# B&R Automation Studio project KeePakST401VersionX (part 3)

#### Types.typ - Exported data types
```iecst
TYPE
	DUT_NDSN_ADI : 	STRUCT
		ui_Size : UINT;
		ui_ADI : UINT;
	END_STRUCT;
	DUT_NDSN_Inventory : 	STRUCT
		b_r_TempCtrl_Board1 : BOOL;
		b_r_TempCtrl_Board2 : BOOL;
		b_r_TempCtrl_Board3 : BOOL;
		b_r_TempCtrl_Board4 : BOOL;
		b_r_OEM_Unit : BOOL;
		b_r_OLED_Unit : BOOL;
		b_r_WIFI_Board : BOOL;
		b_r_Refill_Board : BOOL;
		b_r_Anybus_Board : BOOL;
		b_r_Press_Sensor : BOOL;
		b_r_Press_CtrlValve : BOOL;
		i_r_NumOfTempZones_Internal : INT;
		i_r_NumOfTempZones_External : INT;
		i_r_NumOfMotors : INT;
		i_r_NumOfPumps : INT;
		i_r_NumOfATS : INT;
		i_r_NumOfWebClients : INT;
	END_STRUCT;
	DUT_NDSN_Flex : 	STRUCT
		b_r_SystemReady : BOOL;
		b_r_Fault : BOOL;
		b_r_Alert : BOOL;
		b_r_Stop : BOOL;
		b_r_LostCommunication : BOOL;
		b_w_ClearAlertFault : BOOL;
		b_r_TemperatureReady : BOOL;
		b_r_HeatersOn : BOOL;
		b_r_StandbyOn : BOOL;
		b_r_TemperatureAlert : BOOL;
		b_r_TemperatureFault : BOOL;
		b_r_PumpRunning : BOOL;
		b_r_PumpEnabled : BOOL;
		b_r_Purging : BOOL;
		b_r_TankLevelEmpty : BOOL;
		b_r_TankLevelLow : BOOL;
		b_r_FillSysAlert : BOOL;
		b_r_FillSysFault : BOOL;
		b_r_Filling : BOOL;
		b_r_LidOpen : BOOL;
		b_r_EmptyCalibrated : BOOL;
		b_w_HeatersOnOff : BOOL;
		b_w_StandbyOnOff : BOOL;
		b_w_PumpOnOff : BOOL;
		b_w_Purge : BOOL;
		b_w_ManualFill : BOOL;
		b_w_CalibrateEmpty : BOOL;
		b_w_CalibrateFull : BOOL;
		i_rw_Temp_arr_ZoneSP : ARRAY[0..17]OF INT;
		i_rw_Temp_arr_ZoneActivate : ARRAY[0..17]OF INT;
		i_rw_Temp_GlobalStandbyDelta : INT;
		i_rw_Temp_ManualStandyDuration : INT;
		i_rw_Temp_AutoEnterStandbyTm : INT;
		i_rw_Temp_AutoHeaterOffTime : INT;
		i_rw_Temp_AutoStandbySource : INT;
		i_rw_Temp_UnderTempDelta : INT;
		i_rw_Temp_OverTempDelta : INT;
		i_rw_Temp_Unit : INT;
		i_rw_Temp_GlobalSP : INT;
		i_rw_Temp_GlbalHoseSP : INT;
		i_rw_Temp_GlobalGunSP : INT;
		i_rw_Press_Unit : INT;
		r_rw_Press_SP : REAL;
		r_rw_Press_MaxPressLimit : REAL;
		r_rw_Press_MinPressLimit : REAL;
		r_rw_Press_UnderPressDelta : REAL;
		r_rw_Press_OverPressDelta : REAL;
		i_rw_Press_EnableHighLowAlert : INT;
		i_rw_Press_EnableHydrScale : INT;
		i_rw_Fill_EnableFill : INT;
		i_rw_Fill_TargetFillLevel : INT;
		i_rw_Fill_MaxFillTime : INT;
		i_rw_Fill_AlertStopDelayTime : INT;
		i_rw_Fill_LowLevelThreshold : INT;
		i_rw_Fill_LidOpenAlertTime : INT;
		i_rw_Fill_EmptyStopOnOff : INT;
		i_rw_Pump_AutoPump : INT;
		i_rw_Gen_ReadyDelayTime : INT;
		i_rw_Gen_MassUnit : INT;
		i_r_Temp_arr_ZoneActual : ARRAY[0..17]OF INT;
		i_r_Temp_arr_ZoneStatus : ARRAY[0..17]OF INT;
		r_r_Press_ActualPressure : REAL;
		i_r_Press_SensorAlarm : INT;
		i_r_Fill_TankLevel : INT;
		i_r_Gen_CurrentFaultCode : INT;
		i_r_Gen_SoftwareVersion : INT;
		di_r_Gen_OperationHrs : DINT;
		i_r_Gen_arr_SysInventory : ARRAY[0..3]OF INT;
		st_r_Devices : DUT_NDSN_Inventory;
	END_STRUCT;
END_TYPE
```

#### Lib_PBFlx.fun - Exported functions and function blocks
```iecst
{REDUND_OK} FUNCTION_BLOCK FB_NDSN_MB_PBFlex_CtrlSts (*ProblueFlex Function Block for ModbusTCP _Control& Status*) (*$GROUP=User,$CAT=User,$GROUPICON=User.png,$CATICON=User.png*)
	VAR_INPUT
		IN_b_Enable : {REDUND_UNREPLICABLE} BOOL;
		IN_mb_station : STRING[30];
	END_VAR
	VAR_IN_OUT
		Melter : DUT_NDSN_Flex;
	END_VAR
	VAR
		IO_Input : ARRAY[0..63] OF UINT;
		IO_Output : ARRAY[0..63] OF UINT;
		tm_HeaterOff : TON;
		b_HeaterOff : BOOL;
		b_Temp1 : BOOL;
		b_Temp2 : BOOL;
		b_Temp3 : BOOL;
		b_Temp4 : BOOL;
		b_HeaterOn : BOOL;
		tm_HeaterOnStuck : TON;
		b_HeaterOnStuck : BOOL;
		tm_HeaterOffStuck : TON;
		b_HeaterOffStuck : BOOL;
		tm_PumpOff : TON;
		b_PumpOff : BOOL;
		tm_PumpOnStuck : TON;
		b_PumpOnStuck : BOOL;
		tm_PumpOffStuck : TON;
		b_PumpOffStuck : BOOL;
		tm_StandbyOff : TON;
		b_StandbyOff : BOOL;
		tm_StandbyOnStuck : TON;
		b_StandbyOnStuck : BOOL;
		tm_StandbyOffStuck : TON;
		b_StandbyOffStuck : BOOL;
		b_Temp5 : BOOL;
		b_Temp6 : BOOL;
		b_StandbyOn : BOOL;
		b_PumpOn : BOOL;
		tm_Command : TON;
		b_CommandTimerRising : BOOL;
		b_Init : BOOL;
		tm_Acyc : TON;
		b_read : BOOL;
		ui_AcycRdStatus : UINT;
		i : INT;
		FB_AcycWrite : mbWriteMultipleRegisters;
		FB_AcycRead : mbReadHoldingRegisters;
		ui_AcycWtStatus : UINT;
		i_StartAddressOutput : INT;
		i_StartAddressInput : INT;
		i_datasize : INT;
		i_nrRegisters : UINT;
	END_VAR
END_FUNCTION_BLOCK

{REDUND_OK} FUNCTION_BLOCK FB_NDSN_MB_PBFlex_Process (*ProblueFlex Function Block for ModbusTCP _Process*) (*$GROUP=User,$CAT=User,$GROUPICON=User.png,$CATICON=User.png*)
	VAR_INPUT
		IN_b_Enable : {REDUND_UNREPLICABLE} BOOL;
		IN_mb_station : STRING[30];
	END_VAR
	VAR_IN_OUT
		Melter : DUT_NDSN_Flex;
	END_VAR
	VAR
		IO_Input : ARRAY[0..63] OF UINT;
		IO_Output : ARRAY[0..63] OF UINT;
		b_Init : BOOL;
		tm_Acyc : TON;
		b_read : BOOL;
		st_ADI_List : ARRAY[0..49] OF DUT_NDSN_ADI;
		b_AcycRD_Enable : BOOL;
		b_AcycRD_Done : BOOL;
		b_AcycRD_Tick : BOOL;
		ui_AcycRdStatus_Para : UINT;
		ui_AcycRdStatus : UINT;
		b_AcycRdDnRising : BOOL;
		i : INT;
		arr_ResponseValue : ARRAY[0..17] OF UINT;
		i_ValueIndex : INT;
		i_rwDataSize : INT := 70;
		arr_HMI : ARRAY[0..119] OF UINT;
		arr_HMI_Buffer : ARRAY[0..69] OF UINT;
		arr_HMI_Compare : ARRAY[0..69] OF UINT;
		b_WriteEvent : BOOL;
		arr_WriteIndex : ARRAY[0..30] OF INT;
		i_rwADI_Count : INT := 30;
		i_ADI_Range : INT;
		FB_AcycWrite : mbWriteMultipleRegisters;
		FB_AcycRead_Para : mbReadHoldingRegisters;
		i_ADI_Size : INT := 40;
		i_Index : INT;
		i_Index_Write : INT;
		arr_WriteStartingAddress : ARRAY[0..31] OF INT;
		i_ADI : INT;
		di_Press : UDINT;
		di_Press_psi : UDINT;
		r_Press : REAL;
		r_PressConvert : REAL;
		arr_i_DW_Temp : ARRAY[0..1] OF UINT;
		arr_di_Press_psi : ARRAY[0..1] OF UINT;
		tm_WriteEvent : TON;
		i_CompareIndex : INT;
		b_AcycWT_Done : BOOL;
		b_WriteEventONS : BOOL;
		i_writesize : INT;
		i_arr_WriteBuffer : ARRAY[0..17] OF INT;
		i_Size : INT;
		i_SizeofStruct : INT := 236;
		b_Temp2 : BOOL;
		b_AcycWT_DN_Rising : BOOL;
		b_AcycWT_Start : BOOL;
		b_AcycWT_Rising : BOOL;
		ui_AcycWtStatus : UINT;
		i_wttest : UINT;
		b_AcycWTDnRising : BOOL;
		b_test : BOOL;
		i_StartAddressOutput : INT;
		i_StartAddressInput : INT;
		i_datasize : INT;
		ui_Compare : UINT;
		ui_Ctrl : UINT;
		b_temp1 : BOOL;
		b_Compare : BOOL;
		tm_Compare : TON;
		i_test : INT;
		i_nrRegisters : UINT;
	END_VAR
END_FUNCTION_BLOCK
```

### Program Logical/Simulation/Simulation (IEC)

#### Variables.var
```iecst
VAR
	TON_Test : TON;
END_VAR
```

#### Main.st
```iecst
PROGRAM _INIT

	gIO.DIs.SafetyOK := TRUE;
	gIO.SafetyStatus.SafetyProgramRunning := TRUE;

		TON_Test.PT := T#300ms;

END_PROGRAM

PROGRAM _CYCLIC

	//DetermineDistanceToStopPos(gIO.Encoders.SickSSIPosDegrees,

	TON_Test.IN := NOT TON_Test.Q;
//	TON_Test.PT := T#100ms;
	IF EDGEPOS(TON_Test.Q) THEN
		gIO.Encoders.SickSSIPosDegrees := gIO.Encoders.SickSSIPosDegrees + 1;
	END_IF
	IF (gIO.Encoders.SickSSIPosDegrees > 360) THEN
		gIO.Encoders.SickSSIPosDegrees := 0;
	END_IF
	TON_Test();

END_PROGRAM
```

### Program Logical/ModeControl/ModeControl (IEC) - Copy right:KeePak, B&R  Authors: Nathan Stephens, Jeremy Lee, Cody Jung   Rev:1.0   Date:9-28-17

#### Cyclic.ld - Cyclic code
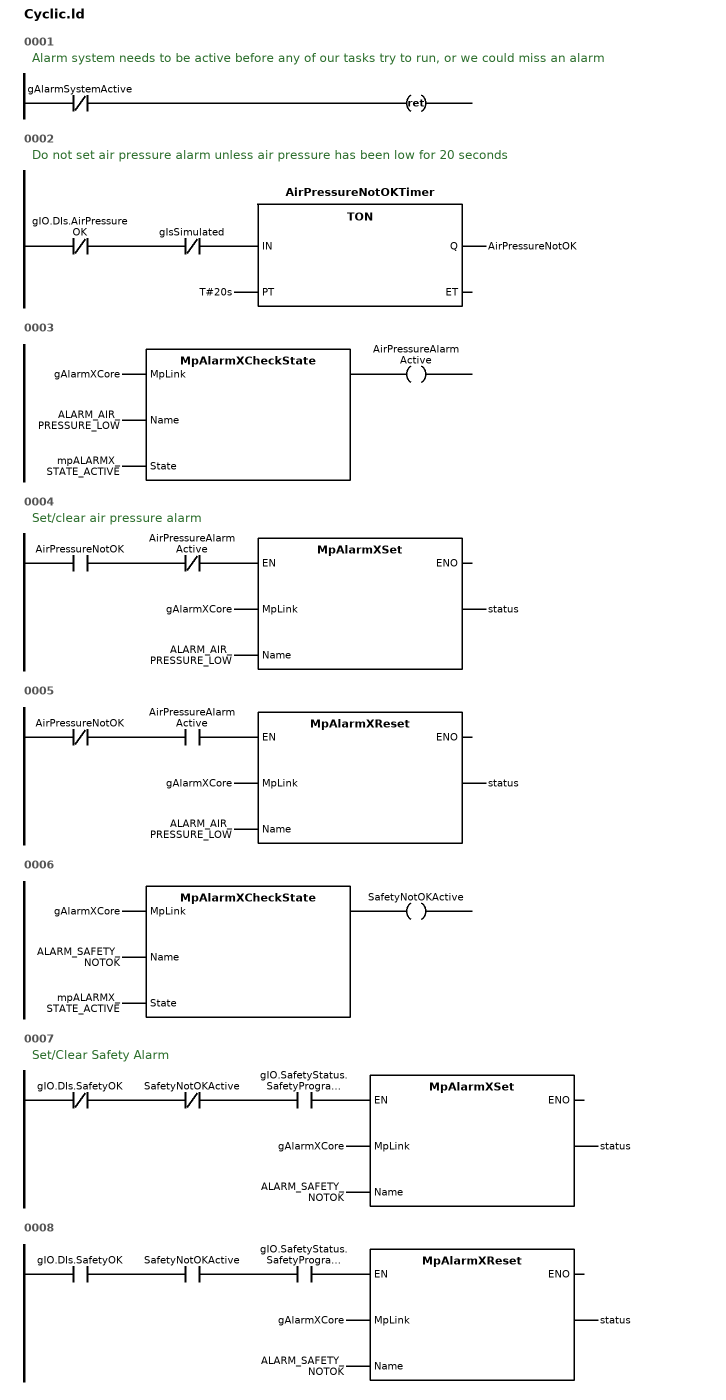
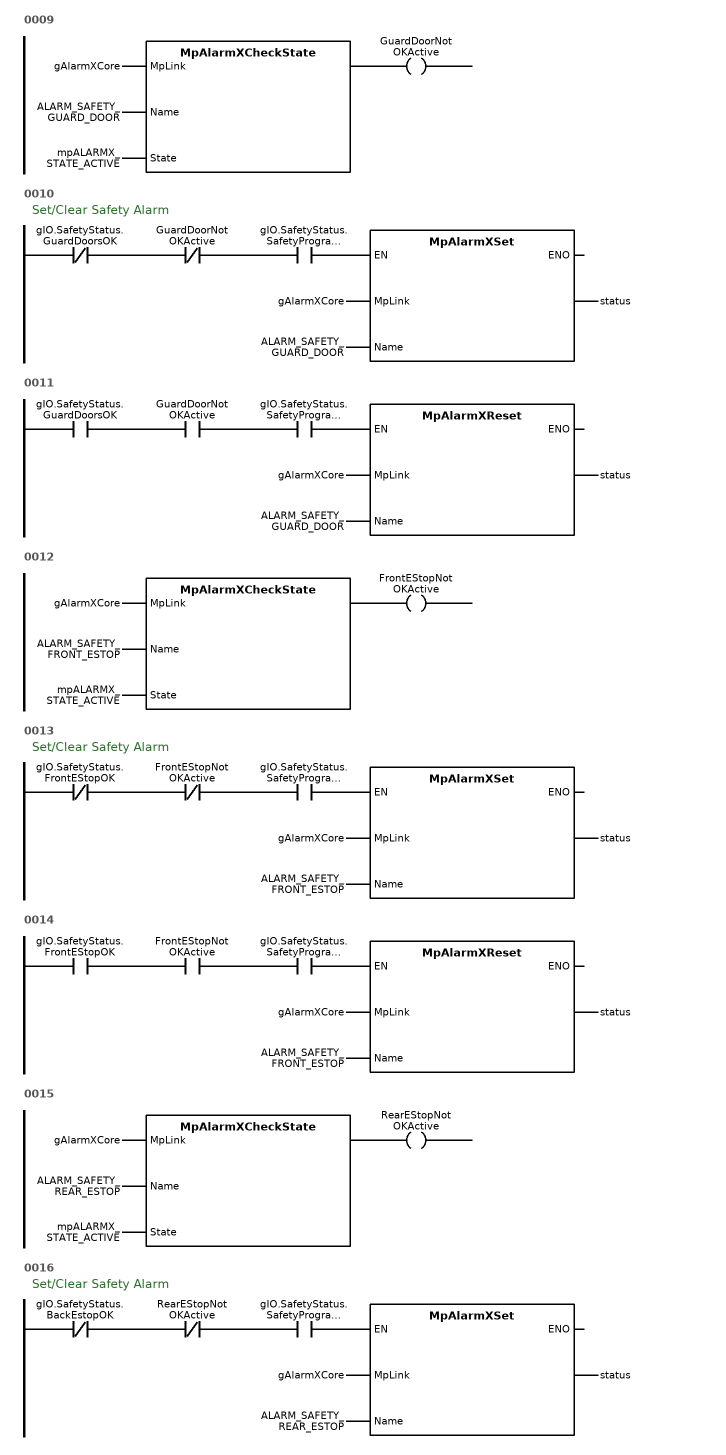
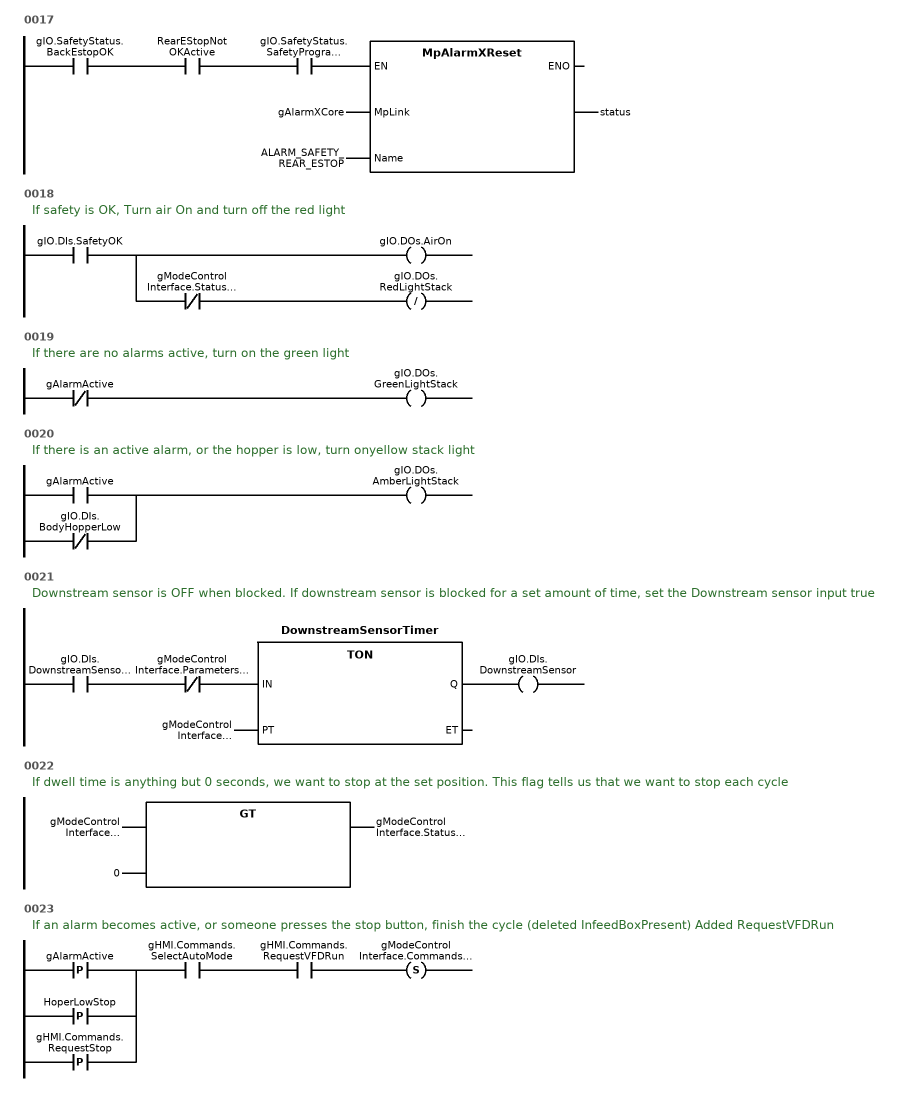
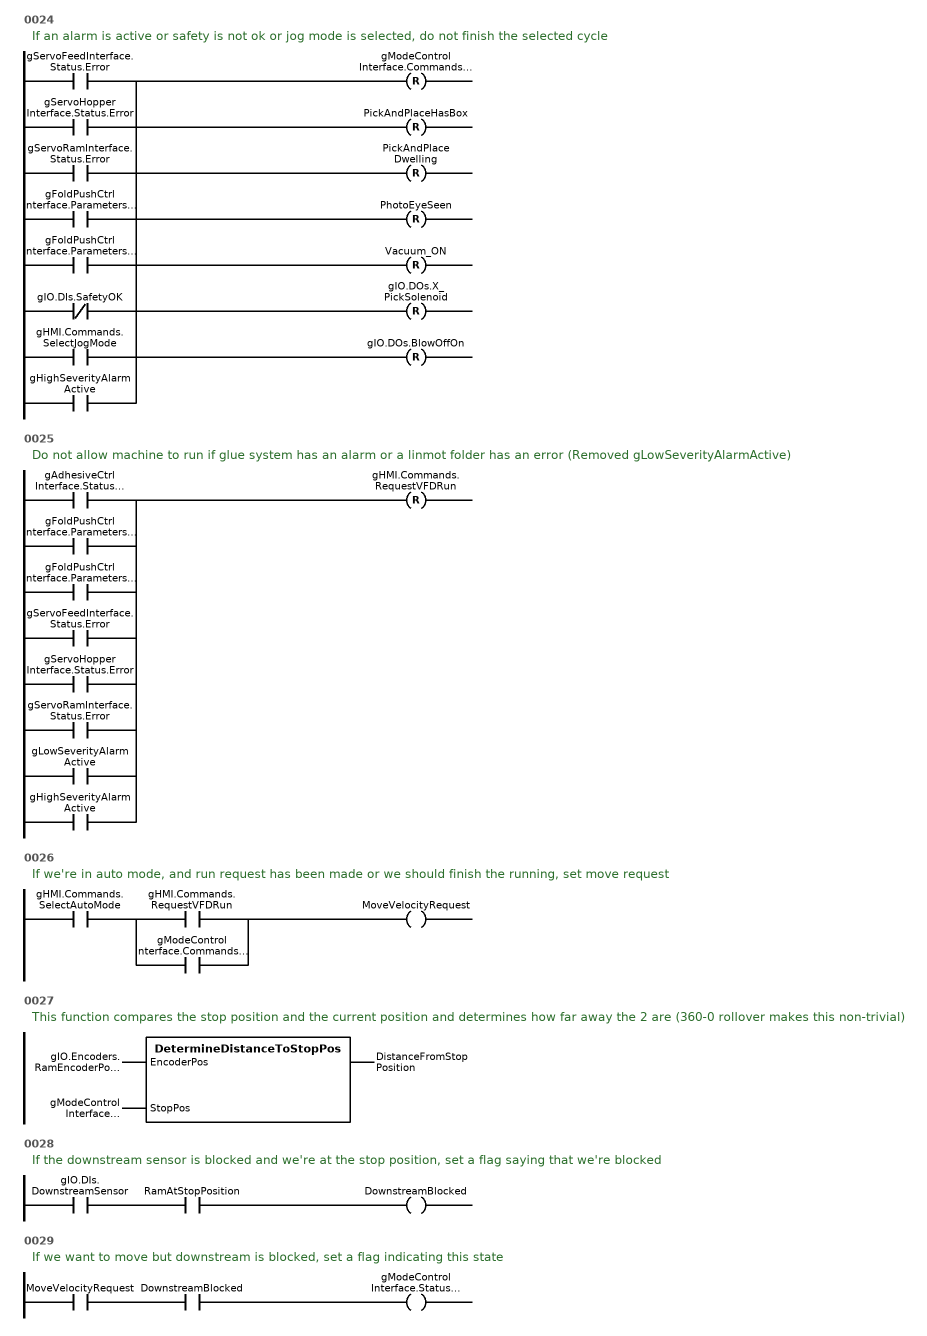
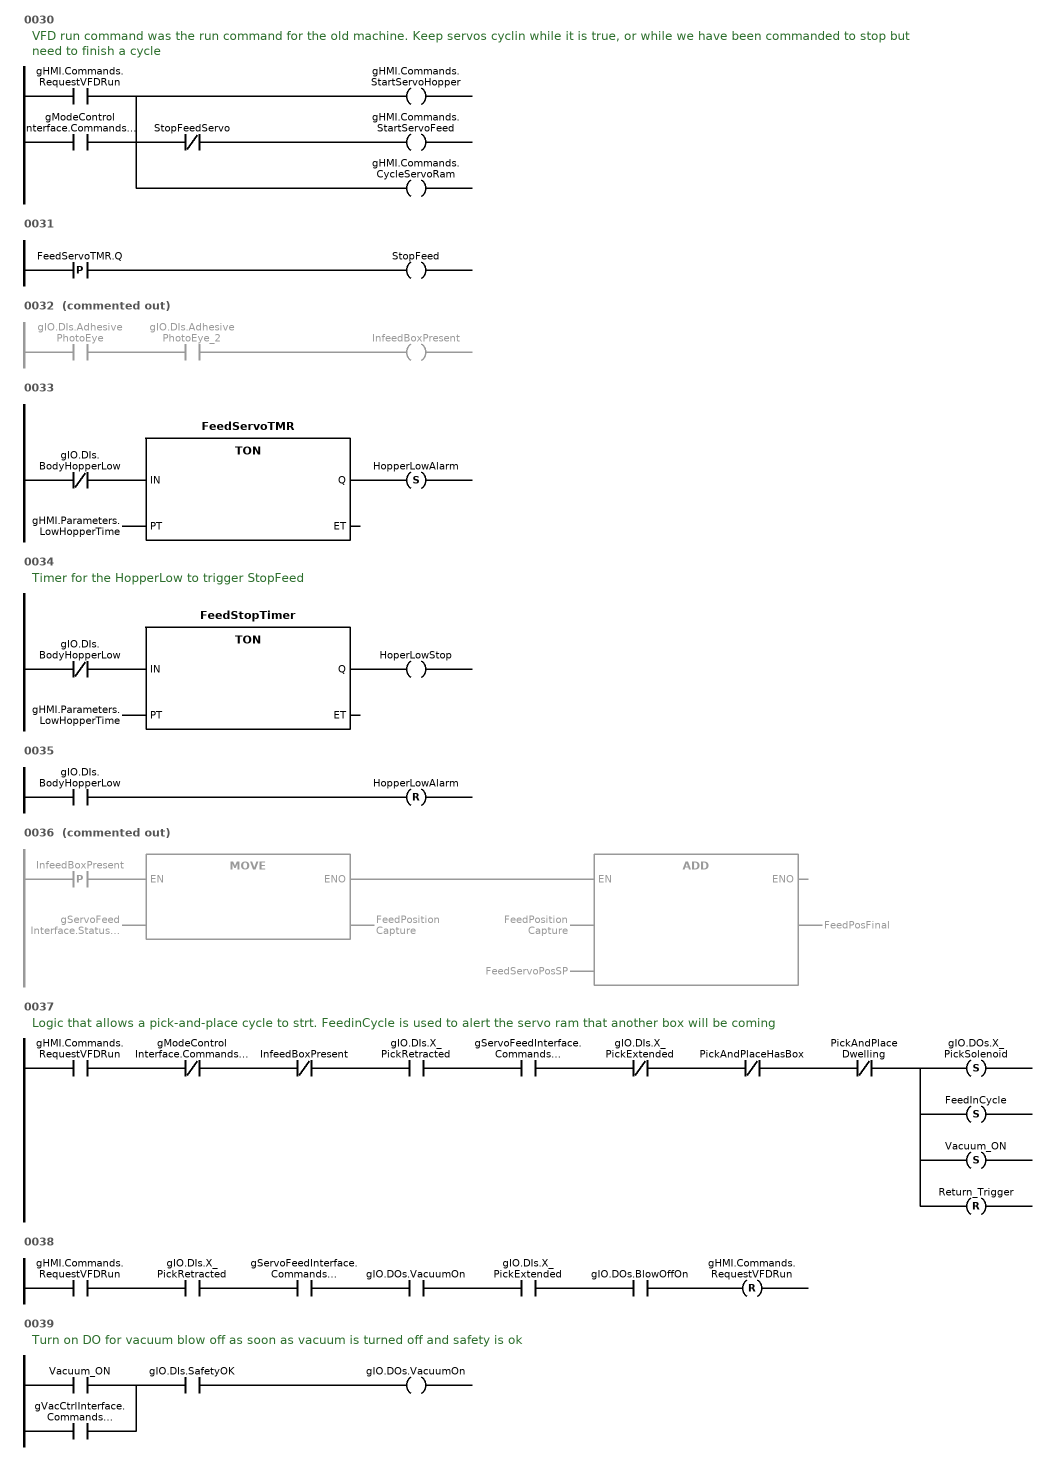
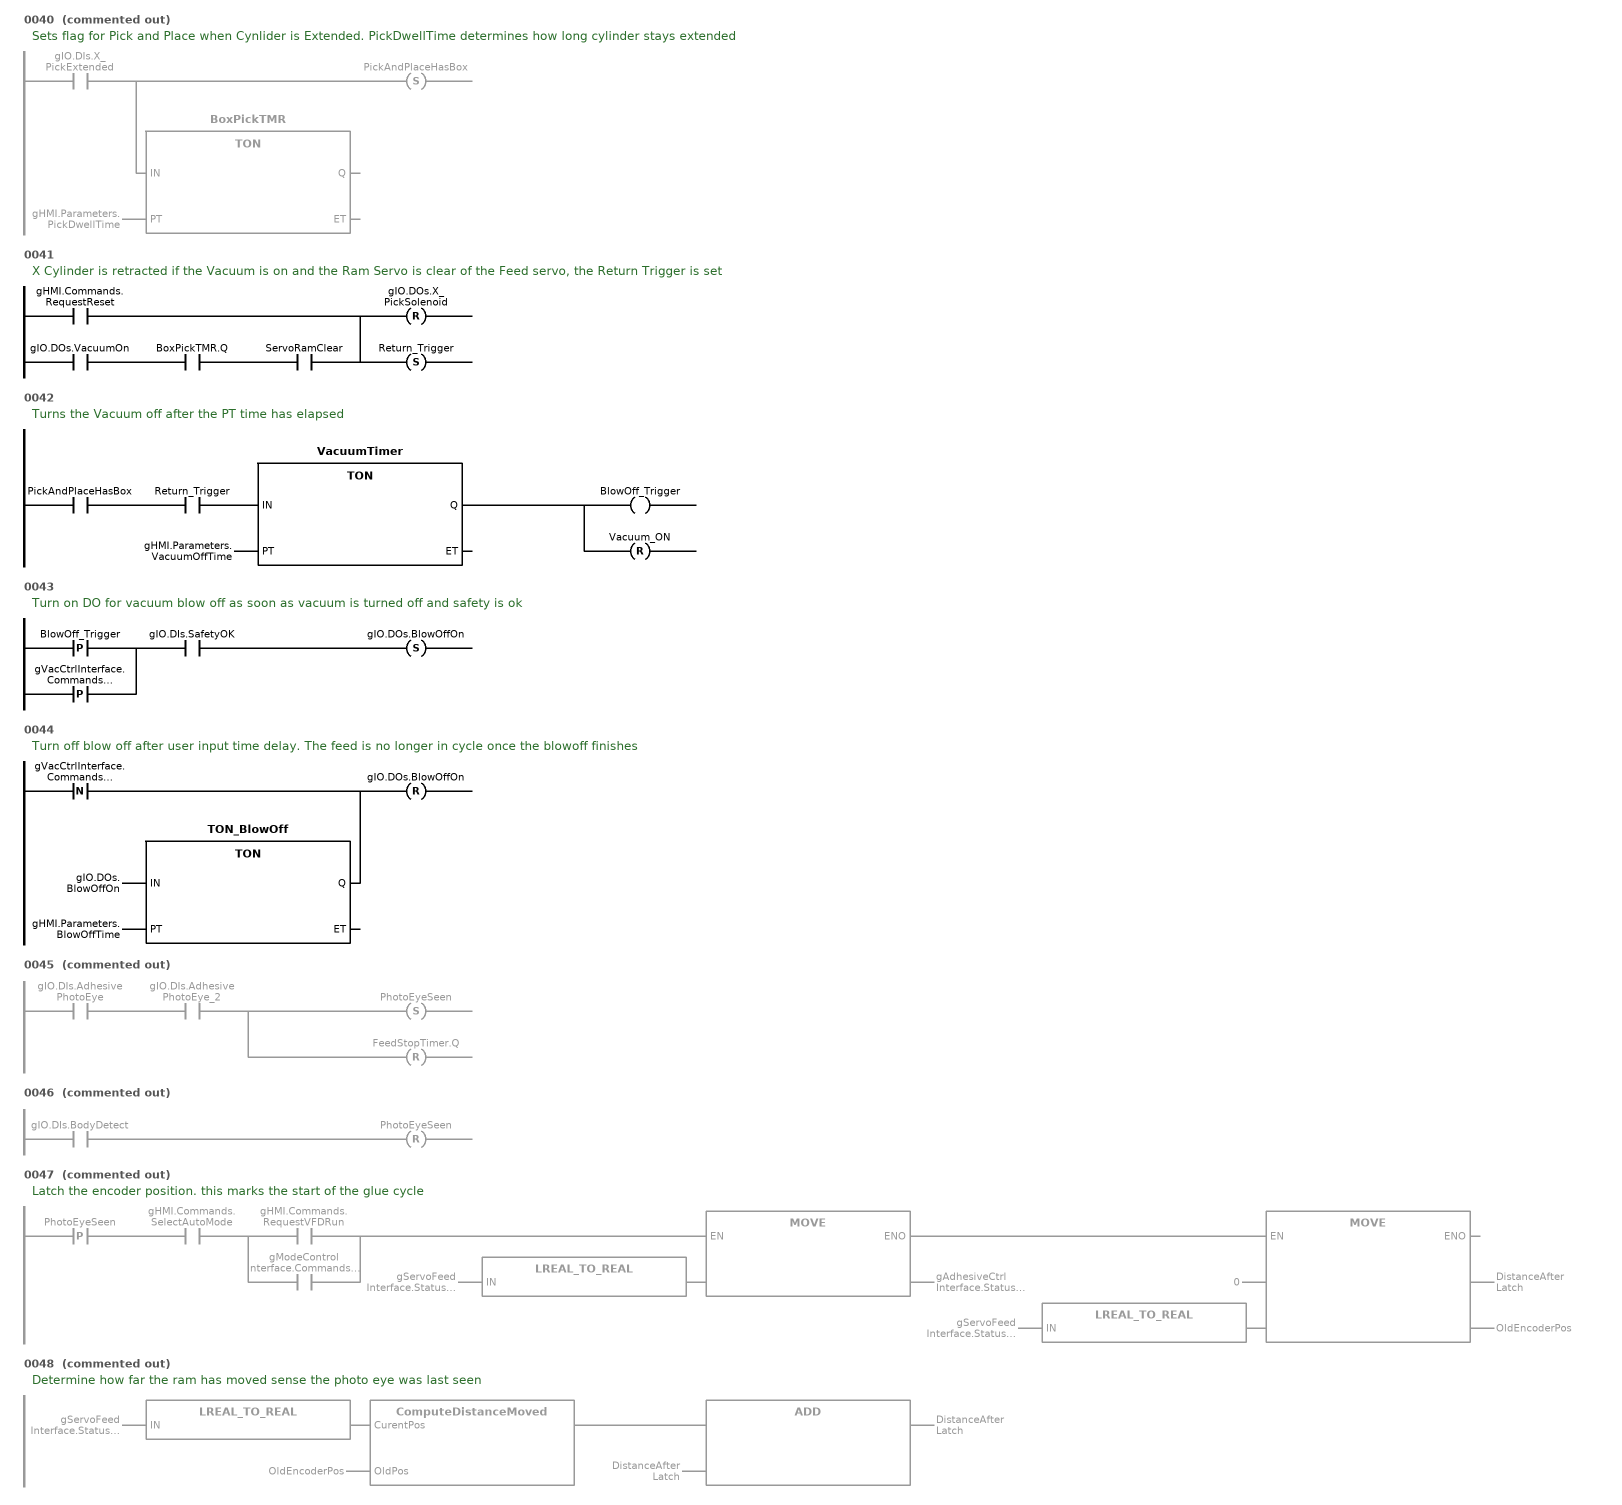
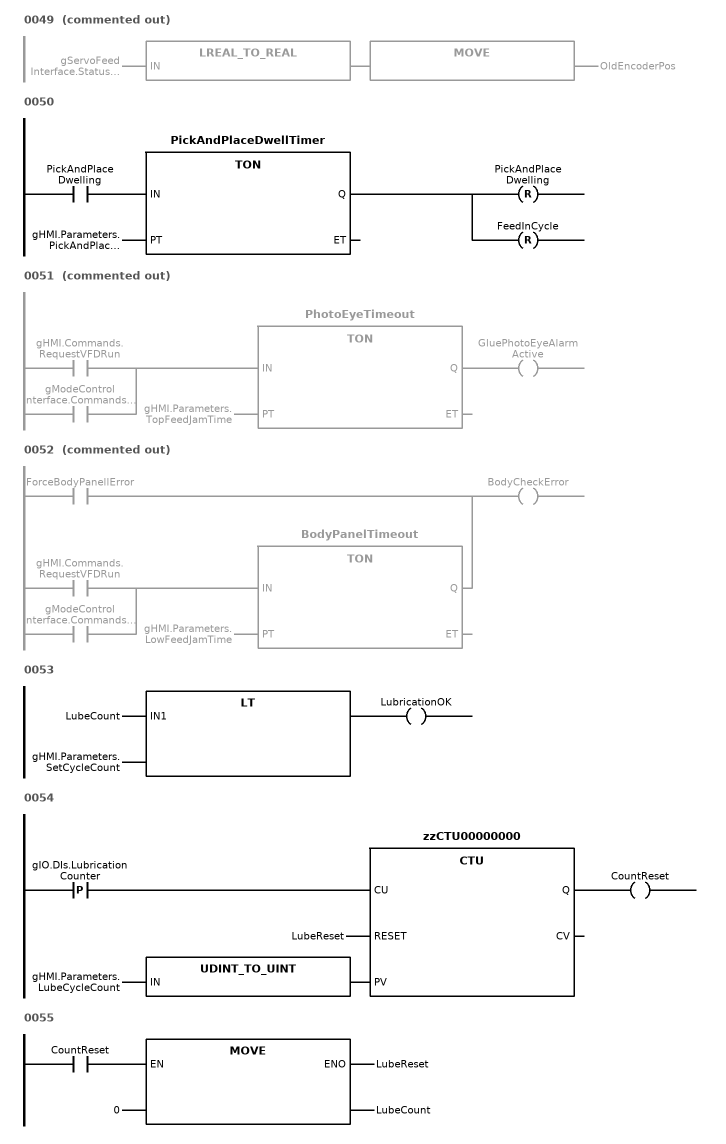
Ladder, written as Structured Text:
```iecst
PROGRAM _CYCLIC
VAR
    _p1 : BOOL;
    _e2 : R_TRIG;
    _e3 : R_TRIG;
    _e4 : R_TRIG;
    _p5 : BOOL;
    _p6 : BOOL;
    _p7 : BOOL;
    _p8 : BOOL;
    _e9 : R_TRIG;
    _e10 : R_TRIG;
    _p11 : BOOL;
    _p12 : BOOL;
    _e13 : R_TRIG;
    _e14 : R_TRIG;
    _e15 : F_TRIG;
    _p16 : BOOL;
    _e17 : R_TRIG;
    _e18 : R_TRIG;
END_VAR
(* Network 1: Alarm system needs to be active before any of our tasks try to run, or we could miss an alarm *)
IF NOT gAlarmSystemActive THEN RETURN; END_IF;

(* Network 2: Do not set air pressure alarm unless air pressure has been low for 20 seconds *)
AirPressureNotOKTimer(IN := NOT gIO.DIs.AirPressureOK AND NOT gIsSimulated, PT := T#20s);
AirPressureNotOK := AirPressureNotOKTimer.Q;

(* Network 3 *)
AirPressureAlarmActive := MpAlarmXCheckState(MpLink := gAlarmXCore, Name := ALARM_AIR_PRESSURE_LOW, State := mpALARMX_STATE_ACTIVE);

(* Network 4: Set/clear air pressure alarm *)
IF AirPressureNotOK AND NOT AirPressureAlarmActive THEN
    status := MpAlarmXSet(MpLink := gAlarmXCore, Name := ALARM_AIR_PRESSURE_LOW);
END_IF;

(* Network 5 *)
IF NOT AirPressureNotOK AND AirPressureAlarmActive THEN
    status := MpAlarmXReset(MpLink := gAlarmXCore, Name := ALARM_AIR_PRESSURE_LOW);
END_IF;

(* Network 6 *)
SafetyNotOKActive := MpAlarmXCheckState(MpLink := gAlarmXCore, Name := ALARM_SAFETY_NOTOK, State := mpALARMX_STATE_ACTIVE);

(* Network 7: Set/Clear Safety Alarm *)
IF NOT gIO.DIs.SafetyOK AND NOT SafetyNotOKActive AND gIO.SafetyStatus.SafetyProgramRunning THEN
    status := MpAlarmXSet(MpLink := gAlarmXCore, Name := ALARM_SAFETY_NOTOK);
END_IF;

(* Network 8 *)
IF gIO.DIs.SafetyOK AND SafetyNotOKActive AND gIO.SafetyStatus.SafetyProgramRunning THEN
    status := MpAlarmXReset(MpLink := gAlarmXCore, Name := ALARM_SAFETY_NOTOK);
END_IF;

(* Network 9 *)
GuardDoorNotOKActive := MpAlarmXCheckState(MpLink := gAlarmXCore, Name := ALARM_SAFETY_GUARD_DOOR, State := mpALARMX_STATE_ACTIVE);

(* Network 10: Set/Clear Safety Alarm *)
IF NOT gIO.SafetyStatus.GuardDoorsOK AND NOT GuardDoorNotOKActive AND gIO.SafetyStatus.SafetyProgramRunning THEN
    status := MpAlarmXSet(MpLink := gAlarmXCore, Name := ALARM_SAFETY_GUARD_DOOR);
END_IF;

(* Network 11 *)
IF gIO.SafetyStatus.GuardDoorsOK AND GuardDoorNotOKActive AND gIO.SafetyStatus.SafetyProgramRunning THEN
    status := MpAlarmXReset(MpLink := gAlarmXCore, Name := ALARM_SAFETY_GUARD_DOOR);
END_IF;

(* Network 12 *)
FrontEStopNotOKActive := MpAlarmXCheckState(MpLink := gAlarmXCore, Name := ALARM_SAFETY_FRONT_ESTOP, State := mpALARMX_STATE_ACTIVE);

(* Network 13: Set/Clear Safety Alarm *)
IF NOT gIO.SafetyStatus.FrontEStopOK AND NOT FrontEStopNotOKActive AND gIO.SafetyStatus.SafetyProgramRunning THEN
    status := MpAlarmXSet(MpLink := gAlarmXCore, Name := ALARM_SAFETY_FRONT_ESTOP);
END_IF;

(* Network 14 *)
IF gIO.SafetyStatus.FrontEStopOK AND FrontEStopNotOKActive AND gIO.SafetyStatus.SafetyProgramRunning THEN
    status := MpAlarmXReset(MpLink := gAlarmXCore, Name := ALARM_SAFETY_FRONT_ESTOP);
END_IF;

(* Network 15 *)
RearEStopNotOKActive := MpAlarmXCheckState(MpLink := gAlarmXCore, Name := ALARM_SAFETY_REAR_ESTOP, State := mpALARMX_STATE_ACTIVE);

(* Network 16: Set/Clear Safety Alarm *)
IF NOT gIO.SafetyStatus.BackEstopOK AND NOT RearEStopNotOKActive AND gIO.SafetyStatus.SafetyProgramRunning THEN
    status := MpAlarmXSet(MpLink := gAlarmXCore, Name := ALARM_SAFETY_REAR_ESTOP);
END_IF;

(* Network 17 *)
IF gIO.SafetyStatus.BackEstopOK AND RearEStopNotOKActive AND gIO.SafetyStatus.SafetyProgramRunning THEN
    status := MpAlarmXReset(MpLink := gAlarmXCore, Name := ALARM_SAFETY_REAR_ESTOP);
END_IF;

(* Network 18: If safety is OK, Turn air On and turn off the red light *)
_p1 := gIO.DIs.SafetyOK;
gIO.DOs.AirOn := gIO.DIs.SafetyOK;
gIO.DOs.RedLightStack := NOT (_p1 AND NOT gModeControlInterface.Status.BlissPanelAlarmActive);

(* Network 19: If there are no alarms active, turn on the green light *)
gIO.DOs.GreenLightStack := NOT gAlarmActive;

(* Network 20: If there is an active alarm, or the hopper is low, turn onyellow stack light *)
gIO.DOs.AmberLightStack := gAlarmActive OR NOT gIO.DIs.BodyHopperLow;

(* Network 21: Downstream sensor is OFF when blocked. If downstream sensor is blocked for a set amount of time, set the Downstream sensor input true *)
DownstreamSensorTimer(IN := gIO.DIs.DownstreamSensorRaw AND NOT gModeControlInterface.Parameters.DownstreamIgnored, PT := gModeControlInterface.Parameters.DownstreamTimeout);
gIO.DIs.DownstreamSensor := DownstreamSensorTimer.Q;

(* Network 22: If dwell time is anything but 0 seconds, we want to stop at the set position. This flag tells us that we want to stop each cycle *)
gModeControlInterface.Status.DwellModeEnabled := gModeControlInterface.Parameters.DwellTime > 0;

(* Network 23: If an alarm becomes active, or someone presses the stop button, finish the cycle (deleted InfeedBoxPresent) Added RequestVFDRun *)
_e2(CLK := gAlarmActive);
_e3(CLK := HoperLowStop);
_e4(CLK := gHMI.Commands.RequestStop);
IF (_e2.Q OR _e3.Q OR _e4.Q) AND gHMI.Commands.SelectAutoMode AND gHMI.Commands.RequestVFDRun THEN
    gModeControlInterface.Commands.FinishCycle := TRUE;
END_IF;

(* Network 24: If an alarm is active or safety is not ok or jog mode is selected, do not finish the selected cycle *)
_p5 := gFoldPushCtrlInterface.Parameters.LinMotBotFolder.Status.Error;
_p6 := gFoldPushCtrlInterface.Parameters.LinMotTopFolder.Status.Error;
IF gServoFeedInterface.Status.Error OR gServoHopperInterface.Status.Error OR gServoRamInterface.Status.Error OR _p5 OR _p6 OR NOT gIO.DIs.SafetyOK OR gHMI.Commands.SelectJogMode OR gHighSeverityAlarmActive THEN
    gModeControlInterface.Commands.FinishCycle := FALSE;
    PickAndPlaceHasBox := FALSE;
    PickAndPlaceDwelling := FALSE;
    PhotoEyeSeen := FALSE;
    Vacuum_ON := FALSE;
END_IF;
_p7 := NOT gIO.DIs.SafetyOK;
IF gServoFeedInterface.Status.Error OR gServoHopperInterface.Status.Error OR gServoRamInterface.Status.Error OR _p5 OR _p6 OR NOT gIO.DIs.SafetyOK OR gHMI.Commands.SelectJogMode OR gHighSeverityAlarmActive THEN
    gIO.DOs.X_PickSolenoid := FALSE;
END_IF;
IF gServoFeedInterface.Status.Error OR gServoHopperInterface.Status.Error OR gServoRamInterface.Status.Error OR _p5 OR _p6 OR _p7 OR gHMI.Commands.SelectJogMode OR gHighSeverityAlarmActive THEN
    gIO.DOs.BlowOffOn := FALSE;
END_IF;

(* Network 25: Do not allow machine to run if glue system has an alarm or a linmot folder has an error (Removed gLowSeverityAlarmActive) *)
IF gAdhesiveCtrlInterface.Status.AlarmActive OR gFoldPushCtrlInterface.Parameters.LinMotBotFolder.Status.Error OR gFoldPushCtrlInterface.Parameters.LinMotTopFolder.Status.Error OR gServoFeedInterface.Status.Error OR gServoHopperInterface.Status.Error OR gServoRamInterface.Status.Error OR gLowSeverityAlarmActive OR gHighSeverityAlarmActive THEN
    gHMI.Commands.RequestVFDRun := FALSE;
END_IF;

(* Network 26: If we're in auto mode, and run request has been made or we should finish the running, set move request *)
MoveVelocityRequest := gHMI.Commands.SelectAutoMode AND (gHMI.Commands.RequestVFDRun OR gModeControlInterface.Commands.FinishCycle);

(* Network 27: This function compares the stop position and the current position and determines how far away the 2 are (360-0 rollover makes this non-trivial) *)
DistanceFromStopPosition := DetermineDistanceToStopPos(EncoderPos := gIO.Encoders.RamEncoderPosDegrees, StopPos := gModeControlInterface.Parameters.StopPosition);

(* Network 28: If the downstream sensor is blocked and we're at the stop position, set a flag saying that we're blocked *)
DownstreamBlocked := gIO.DIs.DownstreamSensor AND RamAtStopPosition;

(* Network 29: If we want to move but downstream is blocked, set a flag indicating this state *)
gModeControlInterface.Status.WaitingOnDownstream := MoveVelocityRequest AND DownstreamBlocked;

(* Network 30: VFD run command was the run command for the old machine. Keep servos cyclin while it is true, or while we have been commanded to stop but need to finish a cycle *)
_p8 := gHMI.Commands.RequestVFDRun;
gHMI.Commands.StartServoHopper := gHMI.Commands.RequestVFDRun OR gModeControlInterface.Commands.FinishCycle;
gHMI.Commands.StartServoFeed := (_p8 OR gModeControlInterface.Commands.FinishCycle) AND NOT StopFeedServo;
gHMI.Commands.CycleServoRam := _p8 OR gModeControlInterface.Commands.FinishCycle;

(* Network 31 *)
_e9(CLK := FeedServoTMR.Q);
StopFeed := _e9.Q;

(* Network 32 *) (* commented out *)
// InfeedBoxPresent := gIO.DIs.AdhesivePhotoEye AND gIO.DIs.AdhesivePhotoEye_2;

(* Network 33 *)
FeedServoTMR(IN := NOT gIO.DIs.BodyHopperLow, PT := gHMI.Parameters.LowHopperTime);
IF FeedServoTMR.Q THEN HopperLowAlarm := TRUE; END_IF;

(* Network 34: Timer for the HopperLow to trigger StopFeed *)
FeedStopTimer(IN := NOT gIO.DIs.BodyHopperLow, PT := gHMI.Parameters.LowHopperTime);
HoperLowStop := FeedStopTimer.Q;

(* Network 35 *)
IF gIO.DIs.BodyHopperLow THEN HopperLowAlarm := FALSE; END_IF;

(* Network 36 *) (* commented out *)
// _e10(CLK := InfeedBoxPresent);
// IF _e10.Q THEN
//     FeedPositionCapture := gServoFeedInterface.Status.ActualPosition;
//     FeedPosFinal := FeedPositionCapture + FeedServoPosSP;
// END_IF;

(* Network 37: Logic that allows a pick-and-place cycle to strt. FeedinCycle is used to alert the servo ram that another box will be coming *)
_p11 := gHMI.Commands.RequestVFDRun AND NOT gModeControlInterface.Commands.FinishCycle AND NOT InfeedBoxPresent AND gIO.DIs.X_PickRetracted AND gServoFeedInterface.Commands.RequestMoveVelocity AND NOT gIO.DIs.X_PickExtended AND NOT PickAndPlaceHasBox AND NOT PickAndPlaceDwelling;
IF _p11 THEN
    gIO.DOs.X_PickSolenoid := TRUE;
    FeedInCycle := TRUE;
    Vacuum_ON := TRUE;
    Return_Trigger := FALSE;
END_IF;

(* Network 38 *)
IF gHMI.Commands.RequestVFDRun AND gIO.DIs.X_PickRetracted AND gServoFeedInterface.Commands.RequestMoveVelocity AND gIO.DOs.VacuumOn AND gIO.DIs.X_PickExtended AND gIO.DOs.BlowOffOn THEN
    gHMI.Commands.RequestVFDRun := FALSE;
END_IF;

(* Network 39: Turn on DO for vacuum blow off as soon as vacuum is turned off and safety is ok *)
gIO.DOs.VacuumOn := (Vacuum_ON OR gVacCtrlInterface.Commands.VenturiOnManual) AND gIO.DIs.SafetyOK;

(* Network 40: Sets flag for Pick and Place when Cynlider is Extended. PickDwellTime determines how long cylinder stays extended *) (* commented out *)
// IF gIO.DIs.X_PickExtended THEN PickAndPlaceHasBox := TRUE; END_IF;
// BoxPickTMR(IN := gIO.DIs.X_PickExtended, PT := gHMI.Parameters.PickDwellTime);

(* Network 41: X Cylinder is retracted if the Vacuum is on and the Ram Servo is clear of the Feed servo, the Return Trigger is set *)
_p12 := gIO.DOs.VacuumOn AND BoxPickTMR.Q AND ServoRamClear;
IF gHMI.Commands.RequestReset OR _p12 THEN
    gIO.DOs.X_PickSolenoid := FALSE;
    Return_Trigger := TRUE;
END_IF;

(* Network 42: Turns the Vacuum off after the PT time has elapsed *)
VacuumTimer(IN := PickAndPlaceHasBox AND Return_Trigger, PT := gHMI.Parameters.VacuumOffTime);
BlowOff_Trigger := VacuumTimer.Q;
IF VacuumTimer.Q THEN Vacuum_ON := FALSE; END_IF;

(* Network 43: Turn on DO for vacuum blow off as soon as vacuum is turned off and safety is ok *)
_e13(CLK := BlowOff_Trigger);
_e14(CLK := gVacCtrlInterface.Commands.BlowOffOnManual);
IF (_e13.Q OR _e14.Q) AND gIO.DIs.SafetyOK THEN gIO.DOs.BlowOffOn := TRUE; END_IF;

(* Network 44: Turn off blow off after user input time delay. The feed is no longer in cycle once the blowoff finishes *)
_e15(CLK := gVacCtrlInterface.Commands.BlowOffOnManual);
IF _e15.Q OR TON_BlowOff.Q THEN gIO.DOs.BlowOffOn := FALSE; END_IF;
TON_BlowOff(IN := gIO.DOs.BlowOffOn, PT := gHMI.Parameters.BlowOffTime);

(* Network 45 *) (* commented out *)
// _p16 := gIO.DIs.AdhesivePhotoEye AND gIO.DIs.AdhesivePhotoEye_2;
// IF _p16 THEN
//     PhotoEyeSeen := TRUE;
//     FeedStopTimer.Q := FALSE;
// END_IF;

(* Network 46 *) (* commented out *)
// IF gIO.DIs.BodyDetect THEN PhotoEyeSeen := FALSE; END_IF;

(* Network 47: Latch the encoder position. this marks the start of the glue cycle *) (* commented out *)
// _e17(CLK := PhotoEyeSeen);
// IF _e17.Q AND gHMI.Commands.SelectAutoMode AND (gHMI.Commands.RequestVFDRun OR gModeControlInterface.Commands.FinishCycle) THEN
//     gAdhesiveCtrlInterface.Status.LatchedEncoderPos := LREAL_TO_REAL(gServoFeedInterface.Status.ActualPosition);
//     DistanceAfterLatch := 0;
//     OldEncoderPos := LREAL_TO_REAL(gServoFeedInterface.Status.ActualPosition);
// END_IF;

(* Network 48: Determine how far the ram has moved sense the photo eye was last seen *) (* commented out *)
// DistanceAfterLatch := ComputeDistanceMoved(CurentPos := LREAL_TO_REAL(gServoFeedInterface.Status.ActualPosition), OldPos := OldEncoderPos) + DistanceAfterLatch;

(* Network 49 *) (* commented out *)
// OldEncoderPos := LREAL_TO_REAL(gServoFeedInterface.Status.ActualPosition);

(* Network 50 *)
PickAndPlaceDwellTimer(IN := PickAndPlaceDwelling, PT := gHMI.Parameters.PickAndPlaceDwell);
IF PickAndPlaceDwellTimer.Q THEN
    PickAndPlaceDwelling := FALSE;
    FeedInCycle := FALSE;
END_IF;

(* Network 51 *) (* commented out *)
// PhotoEyeTimeout(IN := gHMI.Commands.RequestVFDRun OR gModeControlInterface.Commands.FinishCycle, PT := gHMI.Parameters.TopFeedJamTime);
// GluePhotoEyeAlarmActive := PhotoEyeTimeout.Q;

(* Network 52 *) (* commented out *)
// BodyCheckError := ForceBodyPanellError OR BodyPanelTimeout.Q;
// BodyPanelTimeout(IN := gHMI.Commands.RequestVFDRun OR gModeControlInterface.Commands.FinishCycle, PT := gHMI.Parameters.LowFeedJamTime);

(* Network 53 *)
LubricationOK := LubeCount < gHMI.Parameters.SetCycleCount;

(* Network 54 *)
_e18(CLK := gIO.DIs.LubricationCounter);
zzCTU00000000(CU := _e18.Q, RESET := LubeReset, PV := UDINT_TO_UINT(gHMI.Parameters.LubeCycleCount));
CountReset := zzCTU00000000.Q;

(* Network 55 *)
IF CountReset THEN LubeCount := 0; END_IF;
LubeReset := CountReset;
END_PROGRAM
```

#### Init.st
```iecst
PROGRAM _INIT

	//asign default values to parameters
	//defaults, not needed
	(*
	gModeControlInterface.Parameters.PiecesPerMinute := 10;
	gModeControlInterface.Parameters.DwellTime := 0; //ms
	gModeControlInterface.Parameters.StopPosition := 0;

	gAdhesiveCtrlInterface.Parameters.AdhesivePatterns[0].DelayDistance[0] := 150;
	gAdhesiveCtrlInterface.Parameters.AdhesivePatterns[1].DelayDistance[0] := 150;
	gAdhesiveCtrlInterface.Parameters.AdhesivePatterns[2].DelayDistance[0] := 150;
	gAdhesiveCtrlInterface.Parameters.AdhesivePatterns[3].DelayDistance[0] := 150;

	gAdhesiveCtrlInterface.Parameters.AdhesivePatterns[0].GlueOnDistance[0] := 32;
	gAdhesiveCtrlInterface.Parameters.AdhesivePatterns[1].GlueOnDistance[0] := 32;
	gAdhesiveCtrlInterface.Parameters.AdhesivePatterns[2].GlueOnDistance[0] := 32;
	gAdhesiveCtrlInterface.Parameters.AdhesivePatterns[3].GlueOnDistance[0] := 32;

	gAdhesiveCtrlInterface.Parameters.AdhesivePatterns[0].DelayDistance[1] := 210;
	gAdhesiveCtrlInterface.Parameters.AdhesivePatterns[1].DelayDistance[1] := 210;
	gAdhesiveCtrlInterface.Parameters.AdhesivePatterns[2].DelayDistance[1] := 210;
	gAdhesiveCtrlInterface.Parameters.AdhesivePatterns[3].DelayDistance[1] := 210;

	gAdhesiveCtrlInterface.Parameters.AdhesivePatterns[0].GlueOnDistance[1] := 32;
	gAdhesiveCtrlInterface.Parameters.AdhesivePatterns[1].GlueOnDistance[1] := 32;
	gAdhesiveCtrlInterface.Parameters.AdhesivePatterns[2].GlueOnDistance[1] := 32;
	gAdhesiveCtrlInterface.Parameters.AdhesivePatterns[3].GlueOnDistance[1] := 32;

	gAdhesiveCtrlInterface.Parameters.AdhesivePatterns[0].DelayDistance[2] := 300;
	gAdhesiveCtrlInterface.Parameters.AdhesivePatterns[1].DelayDistance[2] := 300;
	gAdhesiveCtrlInterface.Parameters.AdhesivePatterns[2].DelayDistance[2] := 300;
	gAdhesiveCtrlInterface.Parameters.AdhesivePatterns[3].DelayDistance[2] := 300;

	gAdhesiveCtrlInterface.Parameters.AdhesivePatterns[0].GlueOnDistance[2] := 32;
	gAdhesiveCtrlInterface.Parameters.AdhesivePatterns[1].GlueOnDistance[2] := 32;
	gAdhesiveCtrlInterface.Parameters.AdhesivePatterns[2].GlueOnDistance[2] := 32;
	gAdhesiveCtrlInterface.Parameters.AdhesivePatterns[3].GlueOnDistance[2] := 32;

	gFoldPushCtrlInterface.Parameters.BottomFolderOnPos := 100;
	gFoldPushCtrlInterface.Parameters.BottomFolderOffPos := 200;
	gFoldPushCtrlInterface.Parameters.TopFolderOnPos := 180;
	gFoldPushCtrlInterface.Parameters.TopFolderOffPos := 300;
	*)

	gPassword;
	gUserLevel;
	gIO;

	//set these DI's true. physical IO will take over once program runs,
	//and we need to make sure we see a falling edge on these IO points so that alarms are reported
	gIO.DIs.SafetyOK := TRUE;
	gIO.SafetyStatus.BackEstopOK := TRUE;
	gIO.SafetyStatus.FrontEStopOK := TRUE;
	gIO.SafetyStatus.GuardDoorsOK := TRUE;
	gIO.DIs.AirPressureOK := TRUE;
	gIO.DIs.VacuumPressureOK := TRUE;
	gIO.DIs.AdhesiveUnitNotFaulted := TRUE;
	gIO.DIs.AdhesiveUnitReady := TRUE;
	gIO.DIs.AdhesiveLevelLow := FALSE;
	gIO.DIs.VacuumTempOK := TRUE;
	gIO.DIs.BodyHopperLow := TRUE;

	gAutoTune := FALSE;
	gCurrentLimitHit := FALSE;

	//PickDwellTime := T#
	gHMI.Parameters.PickDwellTime :=0;
	gHMI.Parameters.PickAndPlaceDwell := 750; //750 ms
	gHMI.Parameters.LowHopperTime := 3000; //3S
	gHMI.Parameters.LowFeedJamTime := 10000; // 3S
	gHMI.Parameters.TopFeedJamTime := 3000; // 3 S
	gHMI.Parameters.VacuumOffTime := 1000; // 1 S
	gHMI.Parameters.DownPulseTime := 1000; // 1 S
	gHMI.Parameters.Y_DelayTime := 500; // 500ms
	gHMI.Parameters.BlowOffTime := 10; // 10ms
	gHMI.Parameters.LubeCycleCount := 5; // 5 cycles
	gHMI.Parameters.SetCycleCount := 25000; // 25000 Ram Servo Cycles

END_PROGRAM
```

#### Types.typ - Local data types
```iecst
TYPE
	BlissSideCheckStates_enum :
		(
		SIDE_CHECK_IDLE,
		SIDE_CHECK_FIRST_CYCLE,
		SIDE_CHECK_LOOK_FOR_EYE,
		SIDE_CHECK_EYE_FOUND,
		SIDE_CHECK_EYE_MISSED
		);
	BlissBodyCheckStates_enum :
		(
		BODY_CHECK_IDLE,
		BODY_CHECK_FIRST_CYCLE,
		BODY_CHECK_LOOK_FOR_EYE,
		BODY_CHECK_EYE_FOUND,
		BODY_CHECK_EYE_MISSED
		);
	State_enum :
		(
		PICKANDPLACE_ERROR := 99,
		PICKANDPLACE_RETURN := 3,
		PICKANDPLACE_DWELL := 2,
		PICKANDPLACE_MOVE_FORWARD := 1,
		PICKANDPLACE_START := 0
		);
END_TYPE
```

#### Variables.var - Local variables
```iecst
VAR
	AirPressureAlarmActive : BOOL;
	AirPressureNotOK : BOOL;
	AirPressureNotOKTimer : TON;
	BlowOff_Pulse : TP;
	BlowOff_Trigger : BOOL;
	BodyCheckError : BOOL;
	BodyCheckErrorActive : BOOL;
	BodyPanelTimeout : TON;
	BoxPickTMR : TON;
	CountReset : BOOL;
	DistanceFromStopPosition : REAL;
	DownstreamBlocked : BOOL;
	DownstreamSensorTimer : TON;
	Dummy : BOOL;
	DwellTimer : TON;
	EuchnerSafeResetTimer : TON;
	FeedPosFinal : LREAL;
	FeedPositionCapture : LREAL;
	FeedServoPosSP : LREAL;
	FeedServoTimeout : BOOL;
	FeedServoTMR : TON;
	FeedStopTimer : TON;
	ForceBodyPanellError : BOOL;
	FrontEStopNotOKActive : BOOL;
	GluePhotoEyeAlarmActive : BOOL;
	GuardDoorNotOKActive : BOOL;
	HopperLowAlarm : BOOL;
	InBlissSidePanelCheckWindow : BOOL;
	LubeReset : BOOL;
	MoveVelocityRequest : BOOL;
	OldEncoderPos : REAL;
	PhotoEyeCheckErrorActive : BOOL;
	PhotoEyeTimeout : TON;
	PickAndPlaceDwelling : BOOL;
	PickAndPlaceDwellTimer : TON;
	PickAndPlaceHasBox : BOOL;
	PickDwellTime : TIME;
	RamAtStopPosition : BOOL;
	RamCycleCount : UDINT;
	RearEStopNotOKActive : BOOL;
	Return_Trigger : BOOL;
	SafetyNotOKActive : BOOL;
	SafetyResetRequestTimer : TON;
	ShowModeTimer : TON;
	SideCheckError : BOOL;
	SideCheckErrorActive : BOOL;
	state : State_enum;
	status : UDINT;
	StopFeedServo : BOOL;
	StopPositionDwellExpire : BOOL;
	TON_BlowOff : TON; (*Timer for blow off after vacuum is shut off (user defined time)*)
	TON_RamDelay : TON; (*Timer for the Ram to delay forward motion*)
	VacuumOffTime : TIME;
	VacuumTimer : TON;
	Vacuum_ON : BOOL;
	Y_Delay : TON;
	Y_Down_Pulse : TP;
	Y_Trigger : BOOL;
	LubricationCounter : CTU;
END_VAR
```

### Program Logical/ModeControl/ModeControl_ST (IEC) - Copy right:KeePak, B&R  Authors: Nathan Stephens, Jeremy Lee, Cody Jung   Rev:1.0   Date:9-28-17

#### Cyclic1.st
```iecst
PROGRAM _CYCLIC
	(* Insert code here *)

	 //SAFETY CHECKS 0001
    IF NOT gAlarmSystemActive THEN
        RETURN;
    END_IF

    //AIR PRESSURE ON/NOK 0002
    //Do not set air pressure alarm unless air pressure has been low for 20 seconds
    AirPressureNotOKTimer.PT := T#20s;
    AirPressureNotOKTimer.IN := (NOT gIO.DIs.AirPressureOK AND NOT gIsSimulated);
    AirPressureNotOKTimer();
    AirPressureNotOK         := AirPressureNotOKTimer.Q;

    //MP ALARMX CHECK STATE AIR PRESSURE LOW 0003
    AirPressureAlarmActive := MpAlarmXCheckState(gAlarmXCore, ALARM_AIR_PRESSURE_LOW, mpALARMX_STATE_ACTIVE);

    //MP ALARMX SET/RESET AIR PRESSURE LOW 0004 AND 0005
    //Set/clear air pressure alarm
    IF (AirPressureNotOK AND NOT AirPressureAlarmActive) THEN
        status := MpAlarmXSet(gAlarmXCore,ALARM_AIR_PRESSURE_LOW);
    ELSIF (NOT AirPressureNotOK AND AirPressureAlarmActive) THEN
        status := MpAlarmXReset(gAlarmXCore,ALARM_AIR_PRESSURE_LOW);
    END_IF

    //MP ALARMX CHECK STATE SAFETY OK/NOK 0006
    SafetyNotOKActive := MpAlarmXCheckState(gAlarmXCore, ALARM_SAFETY_NOTOK, mpALARMX_STATE_ACTIVE);

    //MP ALARMX SET/RESET SAFETY OK/NOK 0007 AND 0008
    //Set/Clear Safety Alarm
    IF (NOT gIO.DIs.SafetyOK AND NOT SafetyNotOKActive AND gIO.SafetyStatus.SafetyProgramRunning) THEN
        status := MpAlarmXSet(gAlarmXCore,ALARM_SAFETY_NOTOK);
    ELSIF (gIO.DIs.SafetyOK AND SafetyNotOKActive AND gIO.SafetyStatus.SafetyProgramRunning) THEN
        status := MpAlarmXReset(gAlarmXCore,ALARM_SAFETY_NOTOK);
    END_IF

    //MP ALARMX CHECK STATE GUARD DOOR 0009
    GuardDoorNotOKActive := MpAlarmXCheckState(gAlarmXCore, ALARM_SAFETY_GUARD_DOOR, mpALARMX_STATE_ACTIVE);

    //MP ALARMX SET/RESET GUARD DOORS 0010 AND 0011
    //Set/Clear Safety Alarm
    IF (NOT gIO.SafetyStatus.GuardDoorsOK AND NOT GuardDoorNotOKActive AND gIO.SafetyStatus.SafetyProgramRunning) THEN
        status := MpAlarmXSet(gAlarmXCore,ALARM_SAFETY_GUARD_DOOR);
    ELSIF (gIO.SafetyStatus.GuardDoorsOK AND GuardDoorNotOKActive AND gIO.SafetyStatus.SafetyProgramRunning) THEN
        status := MpAlarmXReset(gAlarmXCore,ALARM_SAFETY_GUARD_DOOR);
    END_IF

    //MP ALARMX CHECK STATE FRONT ESTOP 0012
    FrontEStopNotOKActive := MpAlarmXCheckState(gAlarmXCore, ALARM_SAFETY_FRONT_ESTOP, mpALARMX_STATE_ACTIVE);

    //MP ALARMX SET/RESET FRONT ESTOP 0013 AND 0014
    //Set/Clear Safety Alarm
    IF (NOT gIO.SafetyStatus.FrontEStopOK AND NOT FrontEStopNotOKActive AND gIO.SafetyStatus.SafetyProgramRunning) THEN
        status := MpAlarmXSet(gAlarmXCore,ALARM_SAFETY_FRONT_ESTOP);
    ELSIF (gIO.SafetyStatus.FrontEStopOK AND FrontEStopNotOKActive AND gIO.SafetyStatus.SafetyProgramRunning) THEN
        status := MpAlarmXReset(gAlarmXCore,ALARM_SAFETY_FRONT_ESTOP);
    END_IF

    //MP ALARMX CHECK STATE REAR ESTOP 0015
    RearEStopNotOKActive := MpAlarmXCheckState(gAlarmXCore, ALARM_SAFETY_REAR_ESTOP, mpALARMX_STATE_ACTIVE);

    //MP ALARMX SET/RESET REAR ESTOP 0016 AND 0017
    //Set/Clear Safety Alarm
    IF (NOT gIO.SafetyStatus.BackEstopOK AND NOT RearEStopNotOKActive AND gIO.SafetyStatus.SafetyProgramRunning) THEN
        status := MpAlarmXSet(gAlarmXCore,ALARM_SAFETY_REAR_ESTOP);
    ELSIF (gIO.SafetyStatus.BackEstopOK AND RearEStopNotOKActive AND gIO.SafetyStatus.SafetyProgramRunning) THEN
        status := MpAlarmXReset(gAlarmXCore,ALARM_SAFETY_REAR_ESTOP);
    END_IF

    //TURN AIR ON 0018
    //If safety is OK, Turn air On and turn off the red light
    gIO.DOs.AirOn         := gIO.DIs.SafetyOK;
    gIO.DOs.RedLightStack := NOT (gIO.DIs.SafetyOK AND NOT gModeControlInterface.Status.BlissPanelAlarmActive);

    //NO ALARMS GREEN LIGHT 0019
    //If there are no alarms active, turn on the green light
    gIO.DOs.GreenLightStack := NOT gAlarmActive;

    //ALARM YELLOW LIGHT 0020
    //If there is an active alarm, or the hopper is low, turn on yellow stack light
    gIO.DOs.AmberLightStack := (gAlarmActive OR gIO.DIs.BodyHopperLow);

    //DOWNSTREAM SENSOR TIMER SETUP 0021
    //Downstream sensor is OFF when blocked. If downstream sensor is blocked for a set amount of time, set the Downstream sensor input true
    DownstreamSensorTimer.PT := gModeControlInterface.Parameters.DownstreamTimeout;
    DownstreamSensorTimer.IN := (gIO.DIs.DownstreamSensorRaw AND NOT gModeControlInterface.Parameters.DownstreamIgnored);
    DownstreamSensorTimer();
    gIO.DIs.DownstreamSensor := DownstreamSensorTimer.Q; //Writing to an input, cannot do that

 //   IF DownstreamBlocked THEN
 //       Vacuum_ON := FALSE;
 //       FeedInCycle := FALSE;
 //   END_IF;    //added 02/02/23

    ///Added 02/01/2
    //VaccumStopTimer.PT := gModeControlInterface.Parameters.VaccumStopTime;
    //VaccumStopTimer.IN := (gIO.DIs.DownstreamSensorRaw AND NOT gModeControlInterface.Parameters.DownstreamIgnored);
    //VaccumStopTimer();
    //gIO.DOs.VacuumOn := VaccumStopTimer.Q;

   // Downstream sensor when box moves counts down AND THEN starts the machine Added 01-31-23***
    //DownstreamSensorONTimer.PT := gModeControlInterface.Parameters.DownstreamClear;
    //DownstreamSensorONTimer.IN := (gModeControlInterface.Parameters.DownstreamIgnored AND NOT gIO.DIs.DownstreamSensorRaw);
    //DownstreamSensorONTimer();
    //gIO.DIs.DownstreamSensorON := DownstreamSensorONTimer.Q; //Writing to an input, cannot do that

    //0022 IS THE CYCLE DWEL TIMER. WE ARE LETTING THE P&P DWELL BE THE CYCLE PROCESS

    //FFINISH CYCLE BY PRESSING THE STOP BUTTON 0023
    //If an alarm becomes active, or someone presses the stop button, finish the cycle (deleted InfeedBoxPresent) Added RequestVFDRun
    Rtrig_AlarmActive(CLK:= gAlarmActive);
    Rtrig_HopperLow(CLK  := HoperLowStop);
    Rtrig_RequestStop(CLK:= gHMI.Commands.RequestStop);
    Rtrig_DownstreamBlocked(CLK:= DownstreamBlocked);
    Ftrig_DownstreamBlocked(CLK:= gIO.DIs.DownstreamSensor);
    Rtrig_RequestVFDRun(CLK:= gHMI.Commands.RequestVFDRun);
    IF ((Rtrig_AlarmActive.Q OR Rtrig_HopperLow.Q OR Rtrig_RequestStop.Q) AND gHMI.Commands.SelectAutoMode AND (gHMI.Commands.RequestVFDRun OR StopTriggerByDownstream)) THEN
        gModeControlInterface.Commands.FinishCycle := TRUE;
    END_IF
    IF Rtrig_DownstreamBlocked.Q AND NOT gHMI.Commands.RequestStop THEN
        gHMI.Commands.RequestStop := TRUE;
        //gIO.DOs.VacuumOn := FALSE;  //Added 02/01/23
        StopTriggerByDownstream := TRUE;
    END_IF
    IF Ftrig_DownstreamBlocked.Q AND StopTriggerByDownstream THEN
        gHMI.Commands.RequestVFDRun := TRUE;
        gHMI.Commands.RequestStop := FALSE;
        StopTriggerByDownstream := FALSE;
    END_IF
    IF  Rtrig_RequestVFDRun.Q AND StopTriggerByDownstream THEN
        StopTriggerByDownstream := FALSE;
    END_IF

    //DO NOT FINISH CYCLE OF ANYTHING OTHER THAN STOP BUTTON IS PRESSED 0024
    //If an alarm is active or safety is not ok or jog mode is selected, do not finish the selected cycle
    IF (gServoFeedInterface.Status.Error OR gServoHopperInterface.Status.Error OR gServoRamInterface.Status.Error OR
        gFoldPushCtrlInterface.Parameters.LinMotBotFolder.Status.Error OR gFoldPushCtrlInterface.Parameters.LinMotTopFolder.Status.Error OR
        NOT gIO.DIs.SafetyOK OR gHMI.Commands.SelectJogMode OR gHighSeverityAlarmActive OR BodyCheckError) THEN
        gModeControlInterface.Commands.FinishCycle := FALSE;
        PickAndPlaceHasBox                         := FALSE;
        PickAndPlaceDwelling                       := FALSE;
        PhotoEyeSeen                               := FALSE;
        Vacuum_ON                                  := FALSE;
        gIO.DOs.X_PickSolenoid                     := FALSE;
        gIO.DOs.BlowOffOn                          := FALSE;
        state                                      := PICKANDPLACE_ERROR;
    END_IF

    //DOES NOT LET MACHINE RUN IF GLUE SYSTEM HAS AN ERROR 0025
    //Do not allow machine to run if glue system has an alarm or a linmot folder has an error (Removed gLowSeverityAlarmActive)
    IF (gAdhesiveCtrlInterface.Status.AlarmActive OR gFoldPushCtrlInterface.Parameters.LinMotBotFolder.Status.Error OR gFoldPushCtrlInterface.Parameters.LinMotTopFolder.Status.Error OR
        gServoFeedInterface.Status.Error OR gServoHopperInterface.Status.Error OR gServoRamInterface.Status.Error OR
        gLowSeverityAlarmActive OR gHighSeverityAlarmActive) THEN
        gHMI.Commands.RequestVFDRun := FALSE;
    END_IF

    //AUTO MODE RUN REQUEST FINISH CYCLE 0026
    //If we're in auto mode, and run request has been made or we should finish the running, set move request
    MoveVelocityRequest := (gHMI.Commands.SelectAutoMode AND (gHMI.Commands.RequestVFDRun OR gModeControlInterface.Commands.FinishCycle));

    //RAM POSITION AND STOP POSITION (360-0 ROLLOVER)DetermineDistanceToStopPos 0027
    DistanceFromStopPosition := DetermineDistanceToStopPos(gIO.Encoders.FeedEncoderPos, gModeControlInterface.Parameters.StopPosition);

    //DOWNSTREAM SENSOR BLOCKED 0028
    //If the downstream sensor is blocked and we're at the stop position, set a flag saying that we're blocked
    DownstreamBlocked := (gIO.DIs.DownstreamSensor AND gRamAtStopPosition);

    //MOVE WHEN DOWNSTREAM IS BLOCKED 0029
    //If we want to move but downstream is blocked, set a flag indicating this state
    gModeControlInterface.Status.WaitingOnDownstream := (MoveVelocityRequest AND DownstreamBlocked);

    //KEEPS SERVOS RUNNING TO FINISH CYCLE 0030
    //VFD run command was the run command for the old machine. Keep servos cycling while it is true, or while we have been commanded to stop but need to finish a cycle
    gHMI.Commands.StartServoHopper := (gHMI.Commands.RequestVFDRun OR gModeControlInterface.Commands.FinishCycle);
    gHMI.Commands.StartServoFeed   := ((gHMI.Commands.RequestVFDRun OR gModeControlInterface.Commands.FinishCycle) (*AND NOT DownstreamBlocked*) AND NOT StopFeedServo);
    gHMI.Commands.CycleServoRam    := (gHMI.Commands.RequestVFDRun OR gModeControlInterface.Commands.FinishCycle);

    //RISING EDGE FOR SERVOINPUT SIGNAL 0031
    Rtrig_FeedServoTMR(CLK := FeedServoTMR.Q);
    StopFeed := Rtrig_FeedServoTMR.Q;

    //0032 SERVO RAM TRIGGER SET IN FEED HANDLER. COMMENTED OUT

    //HOPPER LOW ALARM 0033
    FeedServoTMR.IN := gIO.DIs.BodyHopperLow;
    FeedServoTMR.PT := gHMI.Parameters.LowHopperTime;
    FeedServoTMR();
    IF FeedServoTMR.Q THEN
        HopperLowAlarm := TRUE;
    END_IF

    //FEED STOP TIMER 0034
    //Timer for the HopperLow to trigger StopFeed
    FeedStopTimer.IN := gIO.DIs.BodyHopperLow;
    FeedStopTimer.PT := gHMI.Parameters.LowHopperTime;
    FeedStopTimer();
    HoperLowStop     := FeedStopTimer.Q;

    //HOPPER LOW ALARM RESET 0035
    IF NOT gIO.DIs.BodyHopperLow THEN
        HopperLowAlarm := FALSE;
    END_IF

    //FEED FINAL POSITION COUNTER 0036 (COMMENTED OUT, BUT TRANSLATING ANYWAY)
    Rtrig_InfeedBoxPresent(CLK := InfeedBoxPresent);
    IF Rtrig_InfeedBoxPresent.Q THEN
        FeedPositionCapture := gServoFeedInterface.Status.ActualPosition;
        FeedPosFinal        := (FeedPositionCapture + FeedServoPosSP);
    END_IF

    //PICK AND PLACE CYCLE START 0037 AND 0038
    //Logic that allows a pick-and-place cycle to strt. FeedInCycle is used to alert the servo ram that another box will be coming
    //In state machine

    //DO FOR VACUUM BLOW OFF 0039
    // this should stay outside of the state machine
    gIO.DOs.VacuumOn := ((Vacuum_ON OR gVacCtrlInterface.Commands.VenturiOnManual) AND gIO.DIs.SafetyOK);

    //	//VACUUM TIMER AFTER PT ELAPSED 0042
    //	//Turns the Vacuum off after the PT time has elapsed
    //	VacuumTimer.PT := gHMI.Parameters.VacuumOffTime;
    //	VacuumTimer.IN := PickAndPlaceHasBox AND Return_Trigger;
    //	VacuumTimer();
    //	BlowOff_Trigger := VacuumTimer.Q;
    //	IF VacuumTimer.Q THEN
    //		Vacuum_ON := FALSE;
    //	END_IF
    //
    //	//DO FOR BLOWOFF WHEN VACUUM IS TURNED OFF AND SAFETY IS OK 0043
    //	//Turn on DO for vacuum blow off as soon as vacuum is turned off and safety is ok
	//	Rtrig_BlowOffTrigger(CLK := BlowOff_Trigger);

	//the blow-off output will obey the manual button only when it is pressed. The timer below will clear the manual blowoff button
	IF gVacCtrlInterface.Commands.BlowOffOnManual THEN
		gIO.DOs.BlowOffOn := gVacCtrlInterface.Commands.BlowOffOnManual;
	END_IF

//	Rtrig_BlowOffManual(CLK  := gVacCtrlInterface.Commands.BlowOffOnManual);
//
//    IF Rtrig_BlowOffManual.Q AND gIO.DIs.SafetyOK THEN
//        gIO.DOs.BlowOffOn := TRUE;
//    ELSE gIO.DOs.BlowOffOn := FALSE;
//    END_IF
    //
    //	//0044 IS BLOW OFF TIMER THAT WE WANT TO CONVERT INTO A DIRECT OUTPUT
	//	//Turn off blow off after user input time delay. The feed is no longer in cycle once the blowoff finishes
	// I re-enabled this code to make the manual blow off button work. The state machine will control the blowoff during auto mode - JDL 3/15/2023
    TON_BlowOff.PT := gHMI.Parameters.BlowOffTime;
    TON_BlowOff.IN := gVacCtrlInterface.Commands.BlowOffOnManual;
    TON_BlowOff();
    //	Ftrig_BlowOffOnManual(CLK := gVacCtrlInterface.Commands.BlowOffOnManual);
	IF (TON_BlowOff.Q) THEN
		gVacCtrlInterface.Commands.BlowOffOnManual := FALSE;
		gIO.DOs.BlowOffOn := FALSE;
	END_IF
    //==========================================================================================================================================================
    //==========================================================================================================================================================

    //PHOTO EYES SETTING AND RESETTING THE PICK AND PLACE. WANT TO REMOVE THIS AND MAKE THE PICK AND PLACE INDEPENDENT 0045
    IF (gIO.DIs.AdhesivePhotoEye AND gIO.DIs.AdhesivePhotoEye_2) THEN
        PhotoEyeSeen := TRUE;
        //The line that should go here would write to an output, which you cannot do
    END_IF

    //BODY DETECT PHOTO EYE 0046
    IF gIO.DIs.BodyDetect THEN
        PhotoEyeSeen := FALSE;
    END_IF

    //0047
    //Latch the encoder position. this marks the start of the glue cycle
    Rtrig_PhotoEyeSeen(CLK := PhotoEyeSeen);
    IF (Rtrig_PhotoEyeSeen.Q AND gHMI.Commands.SelectAutoMode AND (gHMI.Commands.RequestVFDRun OR gModeControlInterface.Commands.FinishCycle)) THEN
        gAdhesiveCtrlInterface.Status.LatchedEncoderPos := LREAL_TO_REAL(gServoFeedInterface.Status.ActualPosition);
        DistanceAfterLatch                              := 0;
        OldEncoderPos                                   := LREAL_TO_REAL(gServoFeedInterface.Status.ActualPosition);
    END_IF

    //0048
    //Determine how far the ram has moved sense the photo eye was last seen
    DistanceAfterLatch := (ComputeDistanceMoved(LREAL_TO_REAL(gServoFeedInterface.Status.ActualPosition),OldEncoderPos) + DistanceAfterLatch);

    //0049
    OldEncoderPos := LREAL_TO_REAL(gServoFeedInterface.Status.ActualPosition);

    //	//PHOTO EYE TIMEOUT 0051
    //	//If the machine is running, but no box passes the photo eye for TopFeedJamTime amount of time, then raise an alarm
    //	PhotoEyeTimeout.PT      := gHMI.Parameters.TopFeedJamTime;
    //	PhotoEyeTimeout.IN      := ((gHMI.Commands.RequestVFDRun OR gModeControlInterface.Commands.FinishCycle) AND NOT PhotoEyeSeen);
    //	PhotoEyeTimeout();
    //	GluePhotoEyeAlarmActive := PhotoEyeTimeout.Q;

    //BODY PANEL TIMEOUT 0052
    //If the machine is running and a box has passed the photoeyes, but hasn't cleared the photo eye for LowFeedJamTime amount of time, then raise an alarm
    BodyPanelTimeout.PT := gHMI.Parameters.LowFeedJamTime;
    BodyPanelTimeout.IN := ((gHMI.Commands.RequestVFDRun OR gModeControlInterface.Commands.FinishCycle) AND NOT gIO.DIs.BodyDetect);
    BodyPanelTimeout();
    IF BodyPanelTimeout.Q THEN
        BodyCheckError := TRUE;
    ELSIF gHMI.Commands.RequestReset THEN
        BodyCheckError := FALSE;
    END_IF

    //0053 AND 0054 LUBE COUNTER
    LubricationOK := (LubeCount < gHMI.Parameters.SetCycleCount);

    Rtrig_LubricationCounter(CLK := gIO.DIs.LubricationCounter);
    LubricationCounter.CU    := Rtrig_LubricationCounter.Q;
    LubricationCounter.RESET := LubeReset;
    LubricationCounter.PV    := UDINT_TO_UINT(gHMI.Parameters.LubeCycleCount);
    LubricationCounter();
    CountReset               := LubricationCounter.Q;

    //0055 COUNT AND LUBE COUNT RESET
    LubeReset := CountReset;
    IF CountReset THEN
        LubeCount := 0;
    END_IF

    //CASE STATEMENT LAYOUT
    PickAndPlaceDwellTimer.IN := FALSE;

    CASE state OF

        PICKANDPLACE_START:
            //When RequestVFDRun goes high (start is pressed), go to move forward state
            IF (gHMI.Commands.RequestVFDRun AND NOT gModeControlInterface.Commands.FinishCycle AND NOT InfeedBoxPresent AND
                gIO.DIs.X_PickRetracted AND gServoFeedInterface.Commands.RequestMoveVelocity AND NOT gIO.DIs.X_PickExtended AND
                NOT PickAndPlaceHasBox AND NOT PickAndPlaceDwelling) THEN
                state := PICKANDPLACE_MOVE_FORWARD;
            END_IF

        PICKANDPLACE_MOVE_FORWARD:
            //Move forward, and turn vacuum on
            gIO.DOs.X_PickSolenoid := TRUE;
            FeedInCycle            := TRUE;
            Return_Trigger         := FALSE;
            Vacuum_ON              := TRUE;
            //When the P&P has extended, raise the PickAndPlaceHasBox flag and start dwelling
            IF gIO.DIs.X_PickExtended THEN
                PickAndPlaceHasBox := TRUE;
                state := PICKANDPLACE_DWELL;
            END_IF

        PICKANDPLACE_DWELL:
            //Dwell while the P&P is grabbing the box. Once the dwell timer finishes, send the P&P home
            PickAndPlaceDwelling := TRUE;
            PickAndPlaceDwellTimer.IN := TRUE;
            PickAndPlaceDwellTimer.PT := gHMI.Parameters.PickAndPlaceDwell;
            IF PickAndPlaceDwellTimer.Q THEN
                PickAndPlaceDwelling := FALSE;
                gIO.DOs.X_PickSolenoid := FALSE;
                Return_Trigger         := TRUE;
                state:= PICKANDPLACE_BLOWOFF;
            END_IF

        PICKANDPLACE_BLOWOFF:
            //Wait for the P&P to pass sensor 11. When this happens, turn off the vacuum and turn on the BlowOff
            IF gIO.DIs.X_BlowOff THEN
                Vacuum_ON := FALSE;
                gIO.DOs.BlowOffOn := TRUE;
                state:= PICKANDPLACE_RETURN;
            END_IF

        PICKANDPLACE_RETURN:
            //Once the P&P has returned home,turn off the BlowOff and either continue the cyclic movement or stop
            IF gIO.DIs.X_PickRetracted THEN
                gIO.DOs.BlowOffOn := FALSE;
                PickAndPlaceHasBox := FALSE;
                IF gHMI.Commands.RequestVFDRun THEN
                    state := PICKANDPLACE_MOVE_FORWARD;
                ELSE
                    state := PICKANDPLACE_START;
                END_IF
            END_IF

        PICKANDPLACE_ERROR:
            IF (gNumActiveAlarms = 0) THEN
                state := PICKANDPLACE_START;
            END_IF
    END_CASE

    PickAndPlaceDwellTimer();

	END_PROGRAM
```

#### Init.st
```iecst
PROGRAM _INIT

	//asign default values to parameters
	//defaults, not needed
	(*
	gModeControlInterface.Parameters.PiecesPerMinute := 10;
	gModeControlInterface.Parameters.DwellTime := 0; //ms
	gModeControlInterface.Parameters.StopPosition := 0;

	gAdhesiveCtrlInterface.Parameters.AdhesivePatterns[0].DelayDistance[0] := 150;
	gAdhesiveCtrlInterface.Parameters.AdhesivePatterns[1].DelayDistance[0] := 150;
	gAdhesiveCtrlInterface.Parameters.AdhesivePatterns[2].DelayDistance[0] := 150;
	gAdhesiveCtrlInterface.Parameters.AdhesivePatterns[3].DelayDistance[0] := 150;

	gAdhesiveCtrlInterface.Parameters.AdhesivePatterns[0].GlueOnDistance[0] := 32;
	gAdhesiveCtrlInterface.Parameters.AdhesivePatterns[1].GlueOnDistance[0] := 32;
	gAdhesiveCtrlInterface.Parameters.AdhesivePatterns[2].GlueOnDistance[0] := 32;
	gAdhesiveCtrlInterface.Parameters.AdhesivePatterns[3].GlueOnDistance[0] := 32;

	gAdhesiveCtrlInterface.Parameters.AdhesivePatterns[0].DelayDistance[1] := 210;
	gAdhesiveCtrlInterface.Parameters.AdhesivePatterns[1].DelayDistance[1] := 210;
	gAdhesiveCtrlInterface.Parameters.AdhesivePatterns[2].DelayDistance[1] := 210;
	gAdhesiveCtrlInterface.Parameters.AdhesivePatterns[3].DelayDistance[1] := 210;

	gAdhesiveCtrlInterface.Parameters.AdhesivePatterns[0].GlueOnDistance[1] := 32;
	gAdhesiveCtrlInterface.Parameters.AdhesivePatterns[1].GlueOnDistance[1] := 32;
	gAdhesiveCtrlInterface.Parameters.AdhesivePatterns[2].GlueOnDistance[1] := 32;
	gAdhesiveCtrlInterface.Parameters.AdhesivePatterns[3].GlueOnDistance[1] := 32;

	gAdhesiveCtrlInterface.Parameters.AdhesivePatterns[0].DelayDistance[2] := 300;
	gAdhesiveCtrlInterface.Parameters.AdhesivePatterns[1].DelayDistance[2] := 300;
	gAdhesiveCtrlInterface.Parameters.AdhesivePatterns[2].DelayDistance[2] := 300;
	gAdhesiveCtrlInterface.Parameters.AdhesivePatterns[3].DelayDistance[2] := 300;

	gAdhesiveCtrlInterface.Parameters.AdhesivePatterns[0].GlueOnDistance[2] := 32;
	gAdhesiveCtrlInterface.Parameters.AdhesivePatterns[1].GlueOnDistance[2] := 32;
	gAdhesiveCtrlInterface.Parameters.AdhesivePatterns[2].GlueOnDistance[2] := 32;
	gAdhesiveCtrlInterface.Parameters.AdhesivePatterns[3].GlueOnDistance[2] := 32;

	gFoldPushCtrlInterface.Parameters.BottomFolderOnPos := 100;
	gFoldPushCtrlInterface.Parameters.BottomFolderOffPos := 200;
	gFoldPushCtrlInterface.Parameters.TopFolderOnPos := 180;
	gFoldPushCtrlInterface.Parameters.TopFolderOffPos := 300;
	*)

	gPassword;
	gUserLevel;
	gIO;

	//set these DI's true. physical IO will take over once program runs,
	//and we need to make sure we see a falling edge on these IO points so that alarms are reported
	gIO.DIs.SafetyOK := TRUE;
	gIO.SafetyStatus.BackEstopOK := TRUE;
	gIO.SafetyStatus.FrontEStopOK := TRUE;
	gIO.SafetyStatus.GuardDoorsOK := TRUE;
	gIO.DIs.AirPressureOK := TRUE;
	gIO.DIs.VacuumPressureOK := TRUE;
	gIO.DIs.AdhesiveUnitNotFaulted := TRUE;
	gIO.DIs.AdhesiveUnitReady := TRUE;
	gIO.DIs.AdhesiveLevelLow := FALSE;
	gIO.DIs.VacuumTempOK := TRUE;
	gIO.DIs.BodyHopperLow := TRUE;

	gAutoTune := FALSE;
	gCurrentLimitHit := FALSE;

	//PickDwellTime := T#
	gHMI.Parameters.PickDwellTime :=0; //Only Used With Older Style Machines
	gHMI.Parameters.PickAndPlaceDwell := 750; //750ms How Long It Takes To Grab A Box
	gHMI.Parameters.LowHopperTime := 2000; //2S Hopper Low Timer
	gHMI.Parameters.LowFeedJamTime := 3000; // 3S Bottom Photo Eye
	gHMI.Parameters.TopFeedJamTime := 10000; // 10S Top Photo Eyes
	gHMI.Parameters.VacuumOffTime := 1000; // 1S Vacuum Off Time
	gHMI.Parameters.DownPulseTime := 1000; // 1S Only Used On Y Axis Machines
	gHMI.Parameters.Y_DelayTime := 500; // 500ms Only Used On Y Axis Machines
	gHMI.Parameters.BlowOffTime := 100; // 100ms Blow Off and Vacuum Off Trigger
	gHMI.Parameters.LubeCycleCount := 5; // 5 cycles Lube Counter
	gHMI.Parameters.SetCycleCount := 25000; // 25000 Ram Servo Cycles

END_PROGRAM
```

#### Types.typ - Local data types
```iecst
TYPE
	BlissSideCheckStates_enum :
		(
		SIDE_CHECK_IDLE,
		SIDE_CHECK_FIRST_CYCLE,
		SIDE_CHECK_LOOK_FOR_EYE,
		SIDE_CHECK_EYE_FOUND,
		SIDE_CHECK_EYE_MISSED
		);
	BlissBodyCheckStates_enum :
		(
		BODY_CHECK_IDLE,
		BODY_CHECK_FIRST_CYCLE,
		BODY_CHECK_LOOK_FOR_EYE,
		BODY_CHECK_EYE_FOUND,
		BODY_CHECK_EYE_MISSED
		);
	State_enum :
		(
		PICKANDPLACE_ERROR := 99,
		PICKANDPLACE_RETURN := 4,
		PICKANDPLACE_BLOWOFF := 3,
		PICKANDPLACE_DWELL := 2,
		PICKANDPLACE_MOVE_FORWARD := 1,
		PICKANDPLACE_START := 0
		);
END_TYPE
```

#### Variables.var - Local variables
```iecst
VAR
	AirPressureAlarmActive : BOOL;
	AirPressureNotOK : BOOL;
	AirPressureNotOKTimer : TON;
	BlowOff_Pulse : TP;
	BlowOff_Trigger : BOOL;
	BodyCheckError : BOOL;
	BodyCheckErrorActive : BOOL;
	BodyPanelTimeout : TON;
	BoxPickTMR : TON;
	CountReset : BOOL;
	DistanceFromStopPosition : REAL;
	DownstreamBlocked : BOOL;
	DownstreamSensorONTimer : TON;
	DownstreamSensorTimer : TON;
	Dummy : BOOL;
	DwellTimer : TON;
	EuchnerSafeResetTimer : TON;
	FeedPosFinal : LREAL;
	FeedPositionCapture : LREAL;
	FeedServoPosSP : LREAL;
	FeedServoTimeout : BOOL;
	FeedServoTMR : TON;
	FeedStopTimer : TON;
	ForceBodyPanellError : BOOL;
	FrontEStopNotOKActive : BOOL;
	VaccumStopTimer : TON;
END_VAR
VAR CONSTANT
	Ftrig_BlowOffOnManual : F_TRIG := (0); (*Falling edge detection function block for this variable*)
END_VAR
VAR
	Ftrig_DownstreamBlocked : F_TRIG;
	GluePhotoEyeAlarmActive : BOOL;
	GuardDoorNotOKActive : BOOL;
	HopperLowAlarm : BOOL;
	InBlissSidePanelCheckWindow : BOOL;
	LubeReset : BOOL;
	LubricationCounter : CTU;
	MoveVelocityRequest : BOOL;
	OldEncoderPos : REAL;
	PhotoEyeCheckErrorActive : BOOL;
	PhotoEyeTimeout : TON;
	PickAndPlaceDwelling : BOOL;
	PickAndPlaceDwellTimer : TON;
	PickAndPlaceHasBox : BOOL;
	PickDwellTime : TIME;
	RamAtStopPosition : BOOL;
	RamCycleCount : UDINT;
	RearEStopNotOKActive : BOOL;
	Return_Trigger : BOOL;
	Rtrig_AlarmActive : R_TRIG; (*Rising edge detection function block for this variable*)
	Rtrig_BlowOffManual : R_TRIG; (*Rising edge detection function block for this variable*)
	Rtrig_BlowOffTrigger : R_TRIG; (*Rising edge detection function block for this variable*)
	Rtrig_DownstreamBlocked : R_TRIG; (*Rising edge detection function block for this variable*)
	Rtrig_FeedServoTMR : R_TRIG; (*Rising edge detection function block for this variable*)
	Rtrig_HopperLow : R_TRIG; (*Rising edge detection function block for this variable*)
	Rtrig_InfeedBoxPresent : R_TRIG; (*Rising edge detection function block for this variable*)
	Rtrig_LubricationCounter : R_TRIG; (*Rising edge detection function block for this variable*)
	Rtrig_PhotoEyeSeen : R_TRIG; (*Rising edge detection function block for this variable*)
	Rtrig_RequestStop : R_TRIG; (*Rising edge detection function block for this variable*)
	Rtrig_RequestVFDRun : R_TRIG;
	SafetyNotOKActive : BOOL;
	SafetyResetRequestTimer : TON;
	ShowModeTimer : TON;
	SideCheckError : BOOL;
	SideCheckErrorActive : BOOL;
	state : State_enum;
	status : UDINT;
	StopFeedServo : BOOL;
	StopPositionDwellExpire : BOOL;
	StopTriggerByDownstream : BOOL;
	TON_BlowOff : TON; (*Timer for blow off after vacuum is shut off (user defined time)*)
	TON_RamDelay : TON; (*Timer for the Ram to delay forward motion*)
	VacuumOffTime : TIME;
	VacuumTimer : TON;
	Vacuum_ON : BOOL;
	Y_Delay : TON;
	Y_Down_Pulse : TP;
	Y_Trigger : BOOL;
END_VAR
```

### Program Logical/Actuators/AdhesiveControl (IEC)

#### Variables.var
```iecst
VAR
	status : UDINT;
	GlueChannel1 : BOOL;
	GlueChannel2 : BOOL;
	GlueChannel3 : BOOL;
	GlueChannel4 : BOOL;
	AdhesiveUnitReadyAlarmActive : BOOL;
	AdhesiveUnitFaultedAlarmActive : BOOL;
	AdhesiveUnitUseageLowAlarmActive : BOOL;
	AdhesiveUnitLevelLowAlarmActive : BOOL;
	Switches0 : ARRAY[0..MAX_NUM_ONOFF_PATTERNS_M1] OF Switches;
	Switches1 : ARRAY[0..MAX_NUM_ONOFF_PATTERNS_M1] OF Switches;
	Switches2 : ARRAY[0..MAX_NUM_ONOFF_PATTERNS_M1] OF Switches;
	Switches3 : ARRAY[0..MAX_NUM_ONOFF_PATTERNS_M1] OF Switches;
END_VAR
```

#### Cyclic.ld
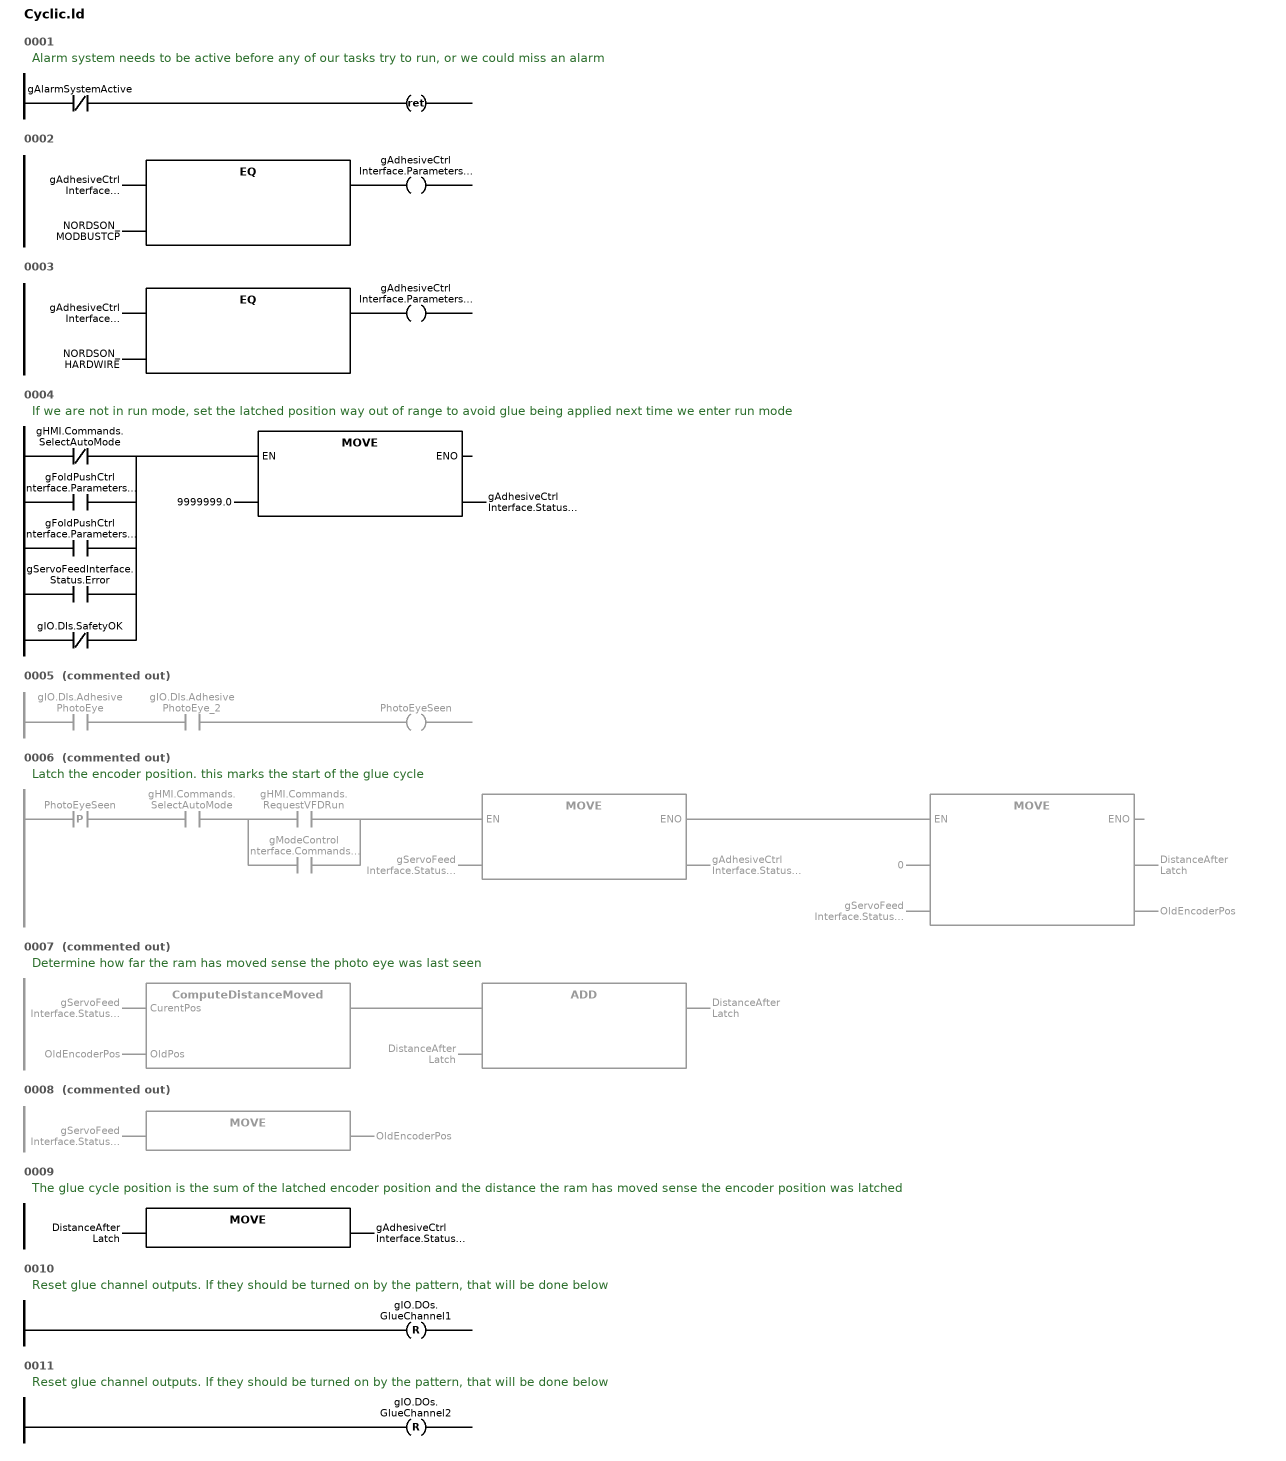
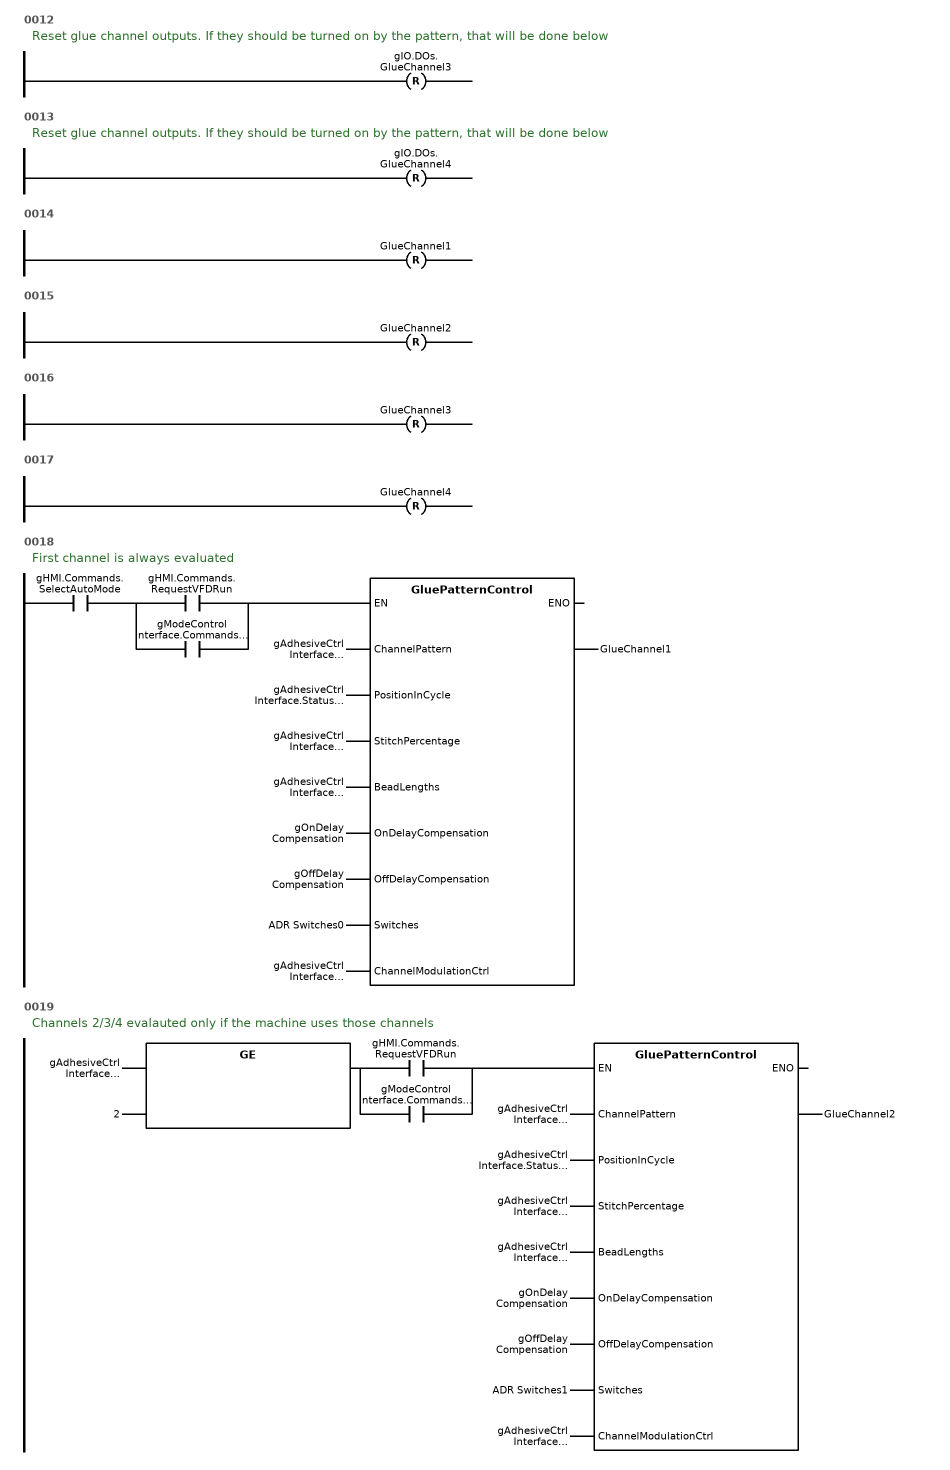
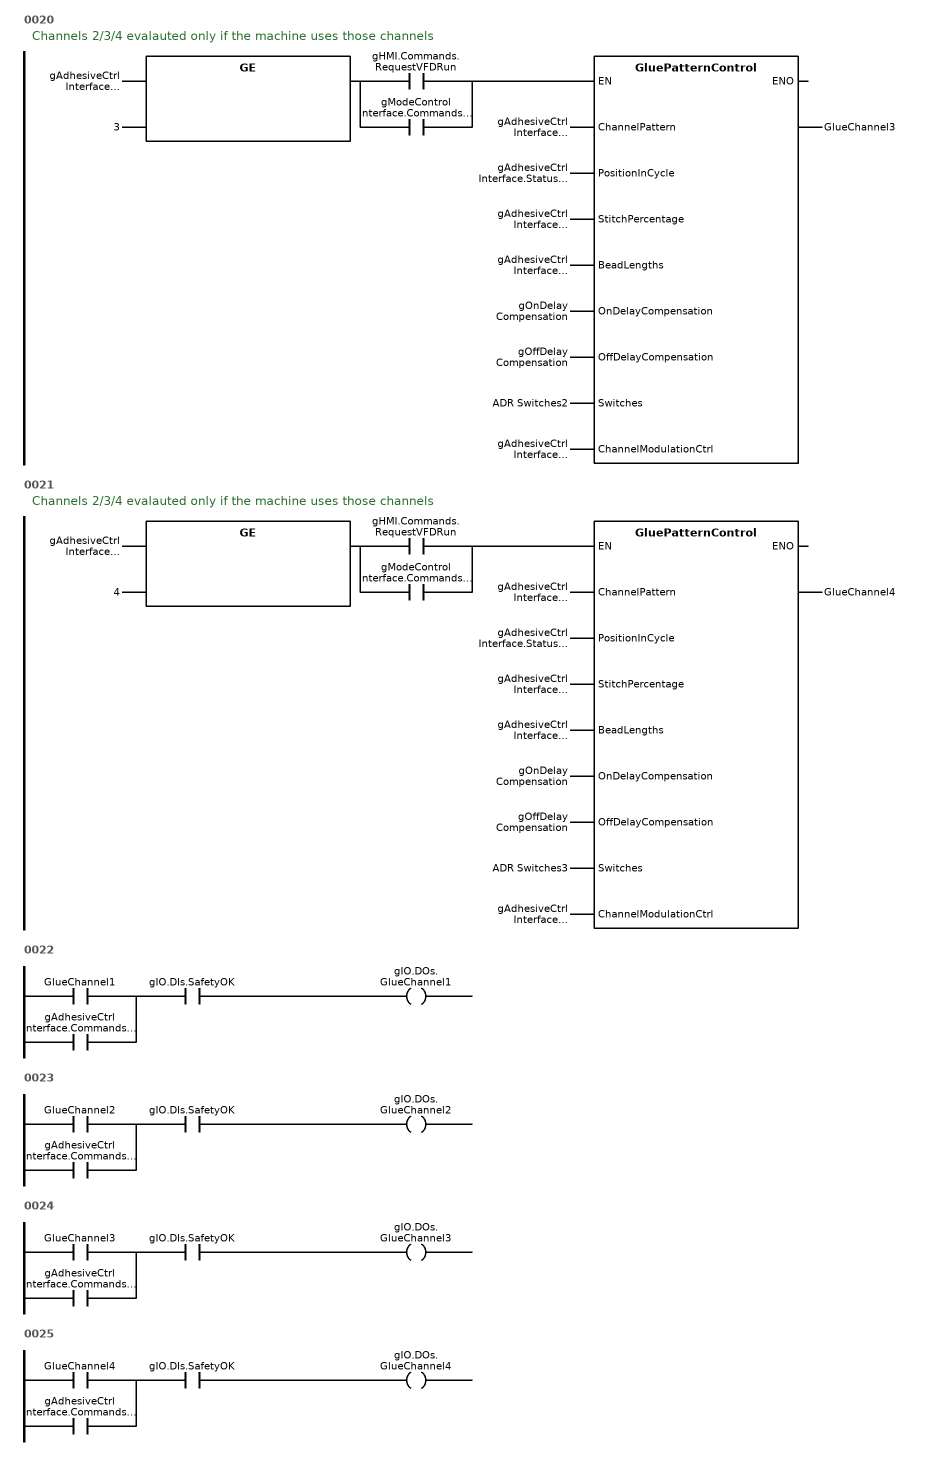
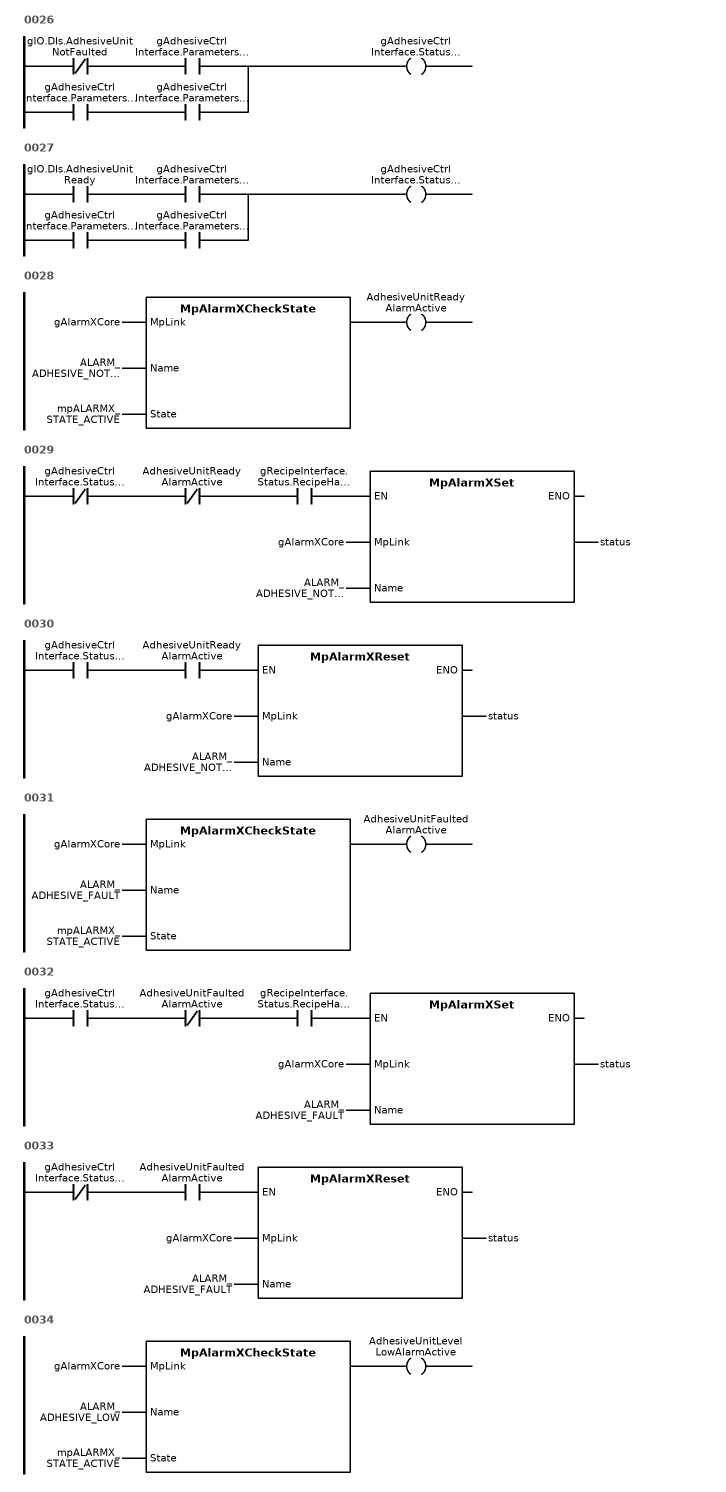
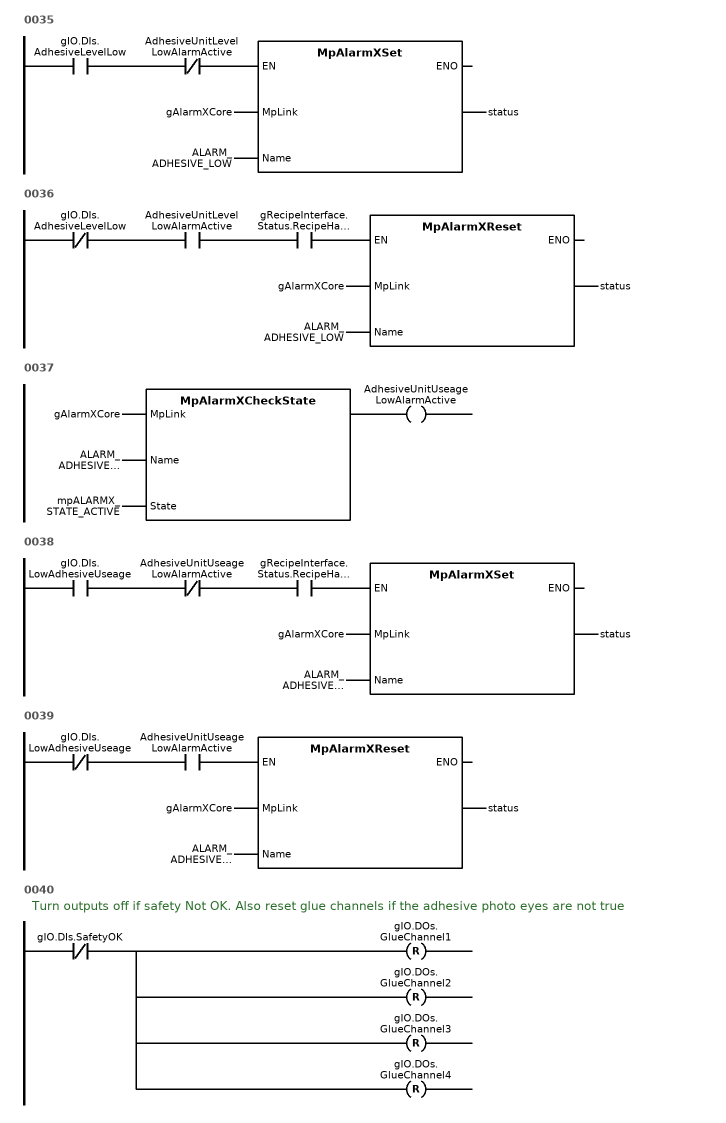
Ladder, written as Structured Text:
```iecst
PROGRAM _CYCLIC
VAR
    _e1 : R_TRIG;
    _t2 : BOOL;
    _t3 : BOOL;
    _t4 : BOOL;
    _p5 : BOOL;
    _p6 : BOOL;
    _p7 : BOOL;
    _p8 : BOOL;
    _p9 : BOOL;
    _p10 : BOOL;
    _p11 : BOOL;
END_VAR
(* Network 1: Alarm system needs to be active before any of our tasks try to run, or we could miss an alarm *)
IF NOT gAlarmSystemActive THEN RETURN; END_IF;

(* Network 2 *)
gAdhesiveCtrlInterface.Parameters.FeedbackIsModbusTCP := gAdhesiveCtrlInterface.Parameters.NordsonFeedbackSelection = NORDSON_MODBUSTCP;

(* Network 3 *)
gAdhesiveCtrlInterface.Parameters.FeedbackIsHardwire := gAdhesiveCtrlInterface.Parameters.NordsonFeedbackSelection = NORDSON_HARDWIRE;

(* Network 4: If we are not in run mode, set the latched position way out of range to avoid glue being applied next time we enter run mode *)
IF NOT gHMI.Commands.SelectAutoMode OR gFoldPushCtrlInterface.Parameters.LinMotBotFolder.Status.Error OR gFoldPushCtrlInterface.Parameters.LinMotTopFolder.Status.Error OR gServoFeedInterface.Status.Error OR NOT gIO.DIs.SafetyOK THEN
    gAdhesiveCtrlInterface.Status.LatchedEncoderPos := 9999999.0;
END_IF;

(* Network 5 *) (* commented out *)
// PhotoEyeSeen := gIO.DIs.AdhesivePhotoEye AND gIO.DIs.AdhesivePhotoEye_2;

(* Network 6: Latch the encoder position. this marks the start of the glue cycle *) (* commented out *)
// _e1(CLK := PhotoEyeSeen);
// IF _e1.Q AND gHMI.Commands.SelectAutoMode AND (gHMI.Commands.RequestVFDRun OR gModeControlInterface.Commands.FinishCycle) THEN
//     gAdhesiveCtrlInterface.Status.LatchedEncoderPos := gServoFeedInterface.Status.ActualPosition;
//     DistanceAfterLatch := 0;
//     OldEncoderPos := gServoFeedInterface.Status.ActualPosition;
// END_IF;

(* Network 7: Determine how far the ram has moved sense the photo eye was last seen *) (* commented out *)
// DistanceAfterLatch := ComputeDistanceMoved(CurentPos := gServoFeedInterface.Status.ActualPosition, OldPos := OldEncoderPos) + DistanceAfterLatch;

(* Network 8 *) (* commented out *)
// OldEncoderPos := gServoFeedInterface.Status.ActualPosition;

(* Network 9: The glue cycle position is the sum of the latched encoder position and the distance the ram has moved sense the encoder position was latched *)
gAdhesiveCtrlInterface.Status.GlueCyclePos := DistanceAfterLatch;

(* Network 10: Reset glue channel outputs. If they should be turned on by the pattern, that will be done below *)
gIO.DOs.GlueChannel1 := FALSE;

(* Network 11: Reset glue channel outputs. If they should be turned on by the pattern, that will be done below *)
gIO.DOs.GlueChannel2 := FALSE;

(* Network 12: Reset glue channel outputs. If they should be turned on by the pattern, that will be done below *)
gIO.DOs.GlueChannel3 := FALSE;

(* Network 13: Reset glue channel outputs. If they should be turned on by the pattern, that will be done below *)
gIO.DOs.GlueChannel4 := FALSE;

(* Network 14 *)
GlueChannel1 := FALSE;

(* Network 15 *)
GlueChannel2 := FALSE;

(* Network 16 *)
GlueChannel3 := FALSE;

(* Network 17 *)
GlueChannel4 := FALSE;

(* Network 18: First channel is always evaluated *)
IF gHMI.Commands.SelectAutoMode AND (gHMI.Commands.RequestVFDRun OR gModeControlInterface.Commands.FinishCycle) THEN
    GlueChannel1 := GluePatternControl(ChannelPattern := gAdhesiveCtrlInterface.Parameters.AdhesivePatterns[0], PositionInCycle := gAdhesiveCtrlInterface.Status.GlueCyclePos, StitchPercentage := gAdhesiveCtrlInterface.Parameters.StitchPercentage, BeadLengths := gAdhesiveCtrlInterface.Parameters.BeadLengths, OnDelayCompensation := gOnDelayCompensation, OffDelayCompensation := gOffDelayCompensation, Switches := ADR(Switches0), ChannelModulationCtrl := gAdhesiveCtrlInterface.Parameters.ChannelModulationCtrl[0]);
END_IF;

(* Network 19: Channels 2/3/4 evalauted only if the machine uses those channels *)
_t2 := gAdhesiveCtrlInterface.Parameters.NumAdhesiveChannels >= 2;
IF _t2 AND (gHMI.Commands.RequestVFDRun OR gModeControlInterface.Commands.FinishCycle) THEN
    GlueChannel2 := GluePatternControl(ChannelPattern := gAdhesiveCtrlInterface.Parameters.AdhesivePatterns[1], PositionInCycle := gAdhesiveCtrlInterface.Status.GlueCyclePos, StitchPercentage := gAdhesiveCtrlInterface.Parameters.StitchPercentage, BeadLengths := gAdhesiveCtrlInterface.Parameters.BeadLengths, OnDelayCompensation := gOnDelayCompensation, OffDelayCompensation := gOffDelayCompensation, Switches := ADR(Switches1), ChannelModulationCtrl := gAdhesiveCtrlInterface.Parameters.ChannelModulationCtrl[1]);
END_IF;

(* Network 20: Channels 2/3/4 evalauted only if the machine uses those channels *)
_t3 := gAdhesiveCtrlInterface.Parameters.NumAdhesiveChannels >= 3;
IF _t3 AND (gHMI.Commands.RequestVFDRun OR gModeControlInterface.Commands.FinishCycle) THEN
    GlueChannel3 := GluePatternControl(ChannelPattern := gAdhesiveCtrlInterface.Parameters.AdhesivePatterns[2], PositionInCycle := gAdhesiveCtrlInterface.Status.GlueCyclePos, StitchPercentage := gAdhesiveCtrlInterface.Parameters.StitchPercentage, BeadLengths := gAdhesiveCtrlInterface.Parameters.BeadLengths, OnDelayCompensation := gOnDelayCompensation, OffDelayCompensation := gOffDelayCompensation, Switches := ADR(Switches2), ChannelModulationCtrl := gAdhesiveCtrlInterface.Parameters.ChannelModulationCtrl[2]);
END_IF;

(* Network 21: Channels 2/3/4 evalauted only if the machine uses those channels *)
_t4 := gAdhesiveCtrlInterface.Parameters.NumAdhesiveChannels >= 4;
IF _t4 AND (gHMI.Commands.RequestVFDRun OR gModeControlInterface.Commands.FinishCycle) THEN
    GlueChannel4 := GluePatternControl(ChannelPattern := gAdhesiveCtrlInterface.Parameters.AdhesivePatterns[3], PositionInCycle := gAdhesiveCtrlInterface.Status.GlueCyclePos, StitchPercentage := gAdhesiveCtrlInterface.Parameters.StitchPercentage, BeadLengths := gAdhesiveCtrlInterface.Parameters.BeadLengths, OnDelayCompensation := gOnDelayCompensation, OffDelayCompensation := gOffDelayCompensation, Switches := ADR(Switches3), ChannelModulationCtrl := gAdhesiveCtrlInterface.Parameters.ChannelModulationCtrl[3]);
END_IF;

(* Network 22 *)
gIO.DOs.GlueChannel1 := (GlueChannel1 OR gAdhesiveCtrlInterface.Commands.PurgeChannel1) AND gIO.DIs.SafetyOK;

(* Network 23 *)
gIO.DOs.GlueChannel2 := (GlueChannel2 OR gAdhesiveCtrlInterface.Commands.PurgeChannel2) AND gIO.DIs.SafetyOK;

(* Network 24 *)
gIO.DOs.GlueChannel3 := (GlueChannel3 OR gAdhesiveCtrlInterface.Commands.PurgeChannel3) AND gIO.DIs.SafetyOK;

(* Network 25 *)
gIO.DOs.GlueChannel4 := (GlueChannel4 OR gAdhesiveCtrlInterface.Commands.PurgeChannel4) AND gIO.DIs.SafetyOK;

(* Network 26 *)
gAdhesiveCtrlInterface.Status.UnitFault := (NOT gIO.DIs.AdhesiveUnitNotFaulted AND gAdhesiveCtrlInterface.Parameters.FeedbackIsHardwire) OR (gAdhesiveCtrlInterface.Parameters.NordsonComms.UnitFaulted AND gAdhesiveCtrlInterface.Parameters.FeedbackIsModbusTCP);

(* Network 27 *)
gAdhesiveCtrlInterface.Status.UnitReady := (gIO.DIs.AdhesiveUnitReady AND gAdhesiveCtrlInterface.Parameters.FeedbackIsHardwire) OR (gAdhesiveCtrlInterface.Parameters.NordsonComms.UnitReady AND gAdhesiveCtrlInterface.Parameters.FeedbackIsModbusTCP);

(* Network 28 *)
AdhesiveUnitReadyAlarmActive := MpAlarmXCheckState(MpLink := gAlarmXCore, Name := ALARM_ADHESIVE_NOT_READY, State := mpALARMX_STATE_ACTIVE);

(* Network 29 *)
_p5 := NOT gAdhesiveCtrlInterface.Status.UnitReady AND NOT AdhesiveUnitReadyAlarmActive AND gRecipeInterface.Status.RecipeHasBeenLoaded;
IF _p5 THEN status := MpAlarmXSet(MpLink := gAlarmXCore, Name := ALARM_ADHESIVE_NOT_READY); END_IF;

(* Network 30 *)
_p6 := gAdhesiveCtrlInterface.Status.UnitReady AND AdhesiveUnitReadyAlarmActive;
IF _p6 THEN status := MpAlarmXReset(MpLink := gAlarmXCore, Name := ALARM_ADHESIVE_NOT_READY); END_IF;

(* Network 31 *)
AdhesiveUnitFaultedAlarmActive := MpAlarmXCheckState(MpLink := gAlarmXCore, Name := ALARM_ADHESIVE_FAULT, State := mpALARMX_STATE_ACTIVE);

(* Network 32 *)
_p7 := gAdhesiveCtrlInterface.Status.UnitFault AND NOT AdhesiveUnitFaultedAlarmActive AND gRecipeInterface.Status.RecipeHasBeenLoaded;
IF _p7 THEN status := MpAlarmXSet(MpLink := gAlarmXCore, Name := ALARM_ADHESIVE_FAULT); END_IF;

(* Network 33 *)
_p8 := NOT gAdhesiveCtrlInterface.Status.UnitFault AND AdhesiveUnitFaultedAlarmActive;
IF _p8 THEN status := MpAlarmXReset(MpLink := gAlarmXCore, Name := ALARM_ADHESIVE_FAULT); END_IF;

(* Network 34 *)
AdhesiveUnitLevelLowAlarmActive := MpAlarmXCheckState(MpLink := gAlarmXCore, Name := ALARM_ADHESIVE_LOW, State := mpALARMX_STATE_ACTIVE);

(* Network 35 *)
IF gIO.DIs.AdhesiveLevelLow AND NOT AdhesiveUnitLevelLowAlarmActive THEN
    status := MpAlarmXSet(MpLink := gAlarmXCore, Name := ALARM_ADHESIVE_LOW);
END_IF;

(* Network 36 *)
_p9 := NOT gIO.DIs.AdhesiveLevelLow AND AdhesiveUnitLevelLowAlarmActive AND gRecipeInterface.Status.RecipeHasBeenLoaded;
IF _p9 THEN status := MpAlarmXReset(MpLink := gAlarmXCore, Name := ALARM_ADHESIVE_LOW); END_IF;

(* Network 37 *)
AdhesiveUnitUseageLowAlarmActive := MpAlarmXCheckState(MpLink := gAlarmXCore, Name := ALARM_ADHESIVE_USEAGE_LOW, State := mpALARMX_STATE_ACTIVE);

(* Network 38 *)
_p10 := gIO.DIs.LowAdhesiveUseage AND NOT AdhesiveUnitUseageLowAlarmActive AND gRecipeInterface.Status.RecipeHasBeenLoaded;
IF _p10 THEN status := MpAlarmXSet(MpLink := gAlarmXCore, Name := ALARM_ADHESIVE_USEAGE_LOW); END_IF;

(* Network 39 *)
IF NOT gIO.DIs.LowAdhesiveUseage AND AdhesiveUnitUseageLowAlarmActive THEN
    status := MpAlarmXReset(MpLink := gAlarmXCore, Name := ALARM_ADHESIVE_USEAGE_LOW);
END_IF;

(* Network 40: Turn outputs off if safety Not OK. Also reset glue channels if the adhesive photo eyes are not true *)
_p11 := NOT gIO.DIs.SafetyOK;
IF NOT gIO.DIs.SafetyOK THEN gIO.DOs.GlueChannel1 := FALSE; END_IF;
IF _p11 THEN
    gIO.DOs.GlueChannel2 := FALSE;
    gIO.DOs.GlueChannel3 := FALSE;
    gIO.DOs.GlueChannel4 := FALSE;
END_IF;
END_PROGRAM
```

#### Init.st
```iecst
PROGRAM _INIT
	(* Insert code here *)
	gAdhesiveCtrlInterface.Parameters.NumAdhesiveChannels := 4;

	DistanceAfterLatch := 99999; //make this large so that the machine doesn't start dispensing glue before it ever sees a photo eye. This will reset to 0 and count up once the photo eye is seen

END_PROGRAM
```

### Program Logical/Actuators/FoldPushControl (IEC)

#### Cyclic.ld - Cyclic code
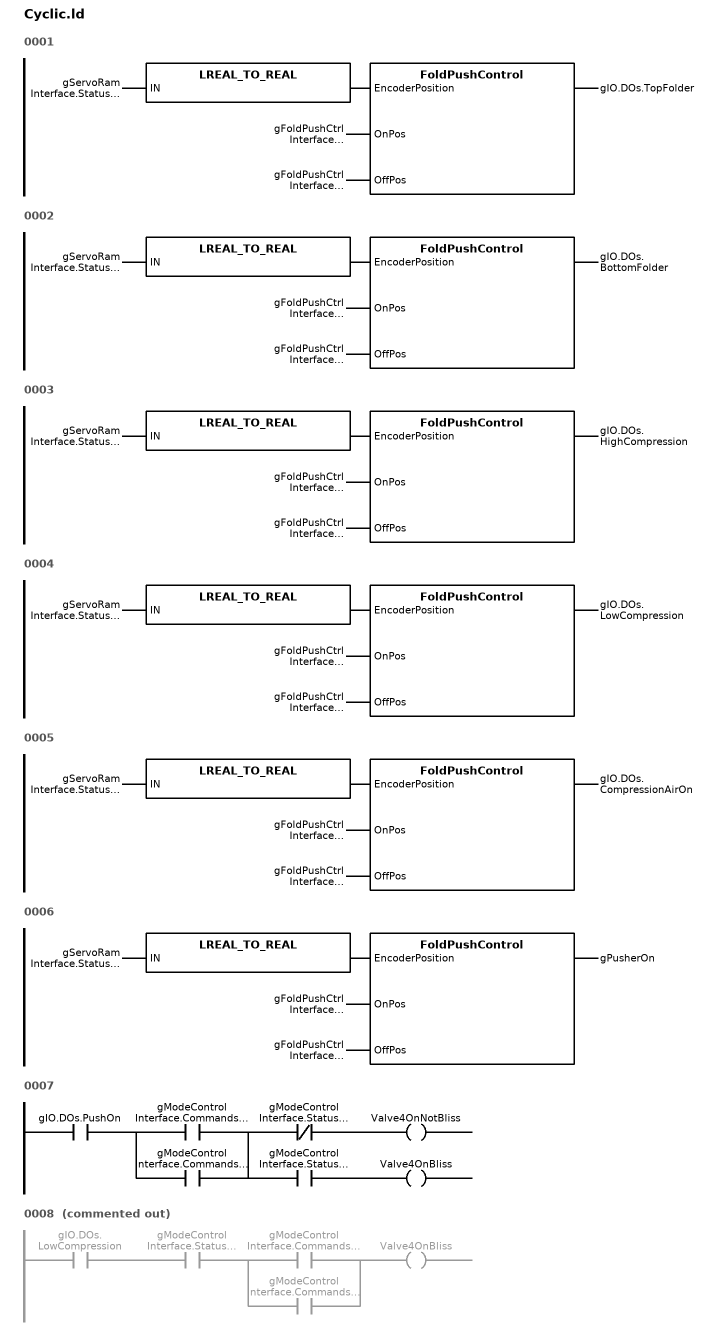
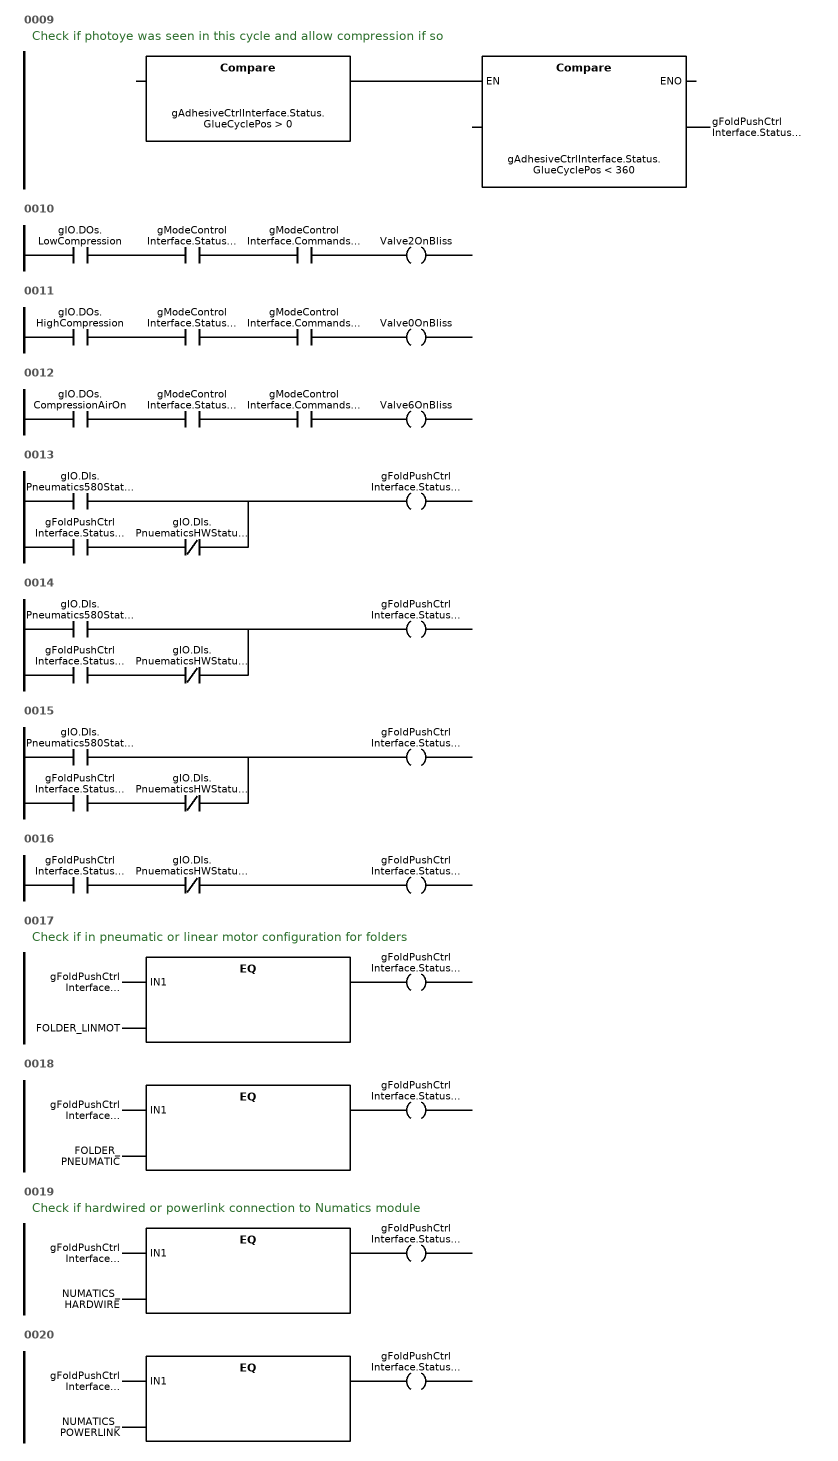
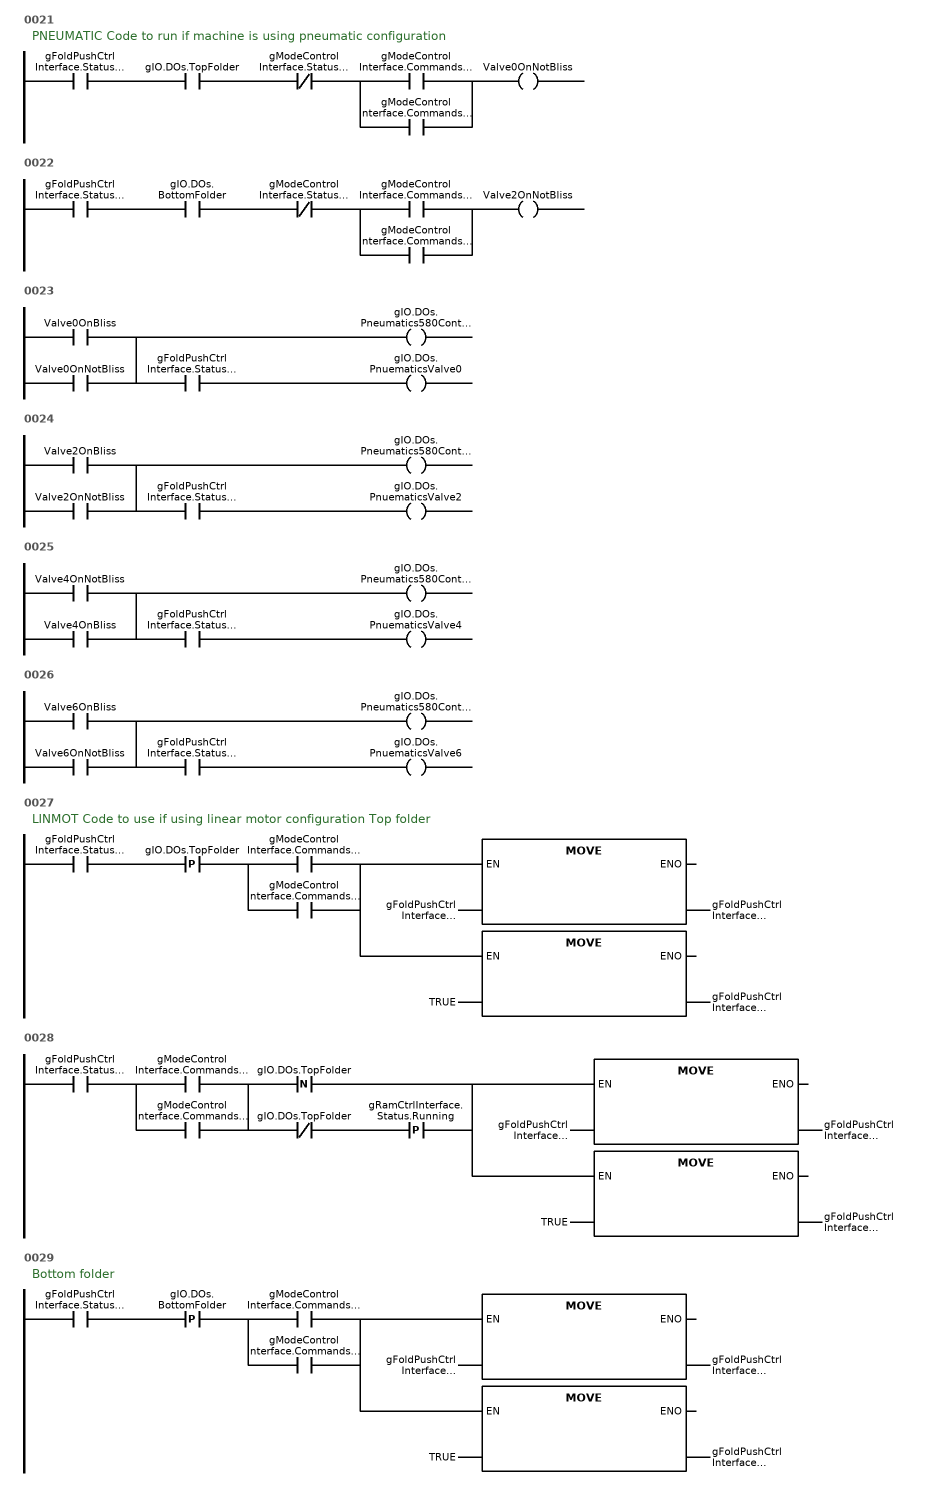
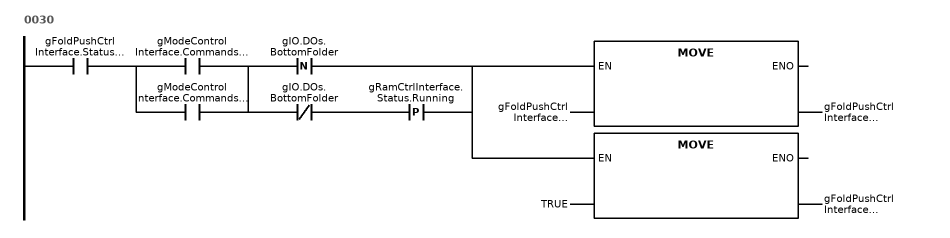
Ladder, written as Structured Text:
```iecst
PROGRAM _CYCLIC
VAR
    _p1 : BOOL;
    _p2 : BOOL;
    _p3 : BOOL;
    _p4 : BOOL;
    _p5 : BOOL;
    _e6 : R_TRIG;
    _p7 : BOOL;
    _p8 : BOOL;
    _p9 : BOOL;
    _p10 : BOOL;
    _p11 : BOOL;
    _e12 : F_TRIG;
    _e13 : R_TRIG;
    _p14 : BOOL;
    _e15 : R_TRIG;
    _p16 : BOOL;
    _p17 : BOOL;
    _p18 : BOOL;
    _p19 : BOOL;
    _p20 : BOOL;
    _e21 : F_TRIG;
    _e22 : R_TRIG;
    _p23 : BOOL;
END_VAR
(* Network 1 *)
gIO.DOs.TopFolder := FoldPushControl(EncoderPosition := LREAL_TO_REAL(gServoRamInterface.Status.ActualPosition), OnPos := gFoldPushCtrlInterface.Parameters.TopFolderOnPos, OffPos := gFoldPushCtrlInterface.Parameters.TopFolderOffPos);

(* Network 2 *)
gIO.DOs.BottomFolder := FoldPushControl(EncoderPosition := LREAL_TO_REAL(gServoRamInterface.Status.ActualPosition), OnPos := gFoldPushCtrlInterface.Parameters.BottomFolderOnPos, OffPos := gFoldPushCtrlInterface.Parameters.BottomFolderOffPos);

(* Network 3 *)
gIO.DOs.HighCompression := FoldPushControl(EncoderPosition := LREAL_TO_REAL(gServoRamInterface.Status.ActualPosition), OnPos := gFoldPushCtrlInterface.Parameters.HighCompressionOnPos, OffPos := gFoldPushCtrlInterface.Parameters.HighCompressionOffPos);

(* Network 4 *)
gIO.DOs.LowCompression := FoldPushControl(EncoderPosition := LREAL_TO_REAL(gServoRamInterface.Status.ActualPosition), OnPos := gFoldPushCtrlInterface.Parameters.LowCompressionOnPos, OffPos := gFoldPushCtrlInterface.Parameters.LowCompressionOffPos);

(* Network 5 *)
gIO.DOs.CompressionAirOn := FoldPushControl(EncoderPosition := LREAL_TO_REAL(gServoRamInterface.Status.ActualPosition), OnPos := gFoldPushCtrlInterface.Parameters.HighCompressionOnPos, OffPos := gFoldPushCtrlInterface.Parameters.LowCompressionOffPos);

(* Network 6 *)
gPusherOn := FoldPushControl(EncoderPosition := LREAL_TO_REAL(gServoRamInterface.Status.ActualPosition), OnPos := gFoldPushCtrlInterface.Parameters.PushOn, OffPos := gFoldPushCtrlInterface.Parameters.PushOff);

(* Network 7 *)
_p1 := gIO.DOs.PushOn AND gModeControlInterface.Commands.SetAutoMode;
_p2 := gIO.DOs.PushOn AND gModeControlInterface.Commands.SetJogMode;
Valve4OnNotBliss := (_p1 OR _p2) AND NOT gModeControlInterface.Status.MachineIsBliss;
Valve4OnBliss := (_p1 OR _p2) AND gModeControlInterface.Status.MachineIsBliss;

(* Network 8 *) (* commented out *)
// _p3 := gIO.DOs.LowCompression AND gModeControlInterface.Status.MachineIsBliss;
// Valve4OnBliss := _p3 AND (gModeControlInterface.Commands.SetAutoMode OR gModeControlInterface.Commands.SetJogMode);

(* Network 9: Check if photoye was seen in this cycle and allow compression if so *)
IF (gAdhesiveCtrlInterface.Status.GlueCyclePos > 0) THEN
    gFoldPushCtrlInterface.Status.CompressionAllowed := gAdhesiveCtrlInterface.Status.GlueCyclePos < 360;
END_IF;

(* Network 10 *)
Valve2OnBliss := gIO.DOs.LowCompression AND gModeControlInterface.Status.MachineIsBliss AND gModeControlInterface.Commands.SetAutoMode;

(* Network 11 *)
Valve0OnBliss := gIO.DOs.HighCompression AND gModeControlInterface.Status.MachineIsBliss AND gModeControlInterface.Commands.SetAutoMode;

(* Network 12 *)
Valve6OnBliss := gIO.DOs.CompressionAirOn AND gModeControlInterface.Status.MachineIsBliss AND gModeControlInterface.Commands.SetAutoMode;

(* Network 13 *)
gFoldPushCtrlInterface.Status.TopFoldValveStatus := gIO.DIs.Pneumatics580StatusWord3.0 OR (gFoldPushCtrlInterface.Status.HardwireConfig AND NOT gIO.DIs.PnuematicsHWStatusV0);

(* Network 14 *)
gFoldPushCtrlInterface.Status.BottomFoldValveStatus := gIO.DIs.Pneumatics580StatusWord3.2 OR (gFoldPushCtrlInterface.Status.HardwireConfig AND NOT gIO.DIs.PnuematicsHWStatusV2);

(* Network 15 *)
gFoldPushCtrlInterface.Status.PushValveStatus := gIO.DIs.Pneumatics580StatusWord3.4 OR (gFoldPushCtrlInterface.Status.HardwireConfig AND NOT gIO.DIs.PnuematicsHWStatusV4);

(* Network 16 *)
gFoldPushCtrlInterface.Status.CompOnValveStatus := gFoldPushCtrlInterface.Status.HardwireConfig AND NOT gIO.DIs.PnuematicsHWStatusV6;

(* Network 17: Check if in pneumatic or linear motor configuration for folders *)
gFoldPushCtrlInterface.Status.LinMotConfig := gFoldPushCtrlInterface.Parameters.FolderTypeSelection = FOLDER_LINMOT;

(* Network 18 *)
gFoldPushCtrlInterface.Status.PneumaticConfig := gFoldPushCtrlInterface.Parameters.FolderTypeSelection = FOLDER_PNEUMATIC;

(* Network 19: Check if hardwired or powerlink connection to Numatics module *)
gFoldPushCtrlInterface.Status.HardwireConfig := gFoldPushCtrlInterface.Parameters.NumaticsTypeSelection = NUMATICS_HARDWIRE;

(* Network 20 *)
gFoldPushCtrlInterface.Status.PowelinkConfig := gFoldPushCtrlInterface.Parameters.NumaticsTypeSelection = NUMATICS_POWERLINK;

(* Network 21: PNEUMATIC Code to run if machine is using pneumatic configuration *)
_p4 := gFoldPushCtrlInterface.Status.PneumaticConfig AND gIO.DOs.TopFolder AND NOT gModeControlInterface.Status.MachineIsBliss;
Valve0OnNotBliss := _p4 AND (gModeControlInterface.Commands.SetAutoMode OR gModeControlInterface.Commands.SetJogMode);

(* Network 22 *)
_p5 := gFoldPushCtrlInterface.Status.PneumaticConfig AND gIO.DOs.BottomFolder AND NOT gModeControlInterface.Status.MachineIsBliss;
Valve2OnNotBliss := _p5 AND (gModeControlInterface.Commands.SetAutoMode OR gModeControlInterface.Commands.SetJogMode);

(* Network 23 *)
gIO.DOs.Pneumatics580ControlWord1.0 := Valve0OnBliss OR Valve0OnNotBliss;
gIO.DOs.PnuematicsValve0 := (Valve0OnBliss OR Valve0OnNotBliss) AND gFoldPushCtrlInterface.Status.HardwireConfig;

(* Network 24 *)
gIO.DOs.Pneumatics580ControlWord1.2 := Valve2OnBliss OR Valve2OnNotBliss;
gIO.DOs.PnuematicsValve2 := (Valve2OnBliss OR Valve2OnNotBliss) AND gFoldPushCtrlInterface.Status.HardwireConfig;

(* Network 25 *)
gIO.DOs.Pneumatics580ControlWord1.4 := Valve4OnNotBliss OR Valve4OnBliss;
gIO.DOs.PnuematicsValve4 := (Valve4OnNotBliss OR Valve4OnBliss) AND gFoldPushCtrlInterface.Status.HardwireConfig;

(* Network 26 *)
gIO.DOs.Pneumatics580ControlWord1.6 := Valve6OnBliss OR Valve6OnNotBliss;
gIO.DOs.PnuematicsValve6 := (Valve6OnBliss OR Valve6OnNotBliss) AND gFoldPushCtrlInterface.Status.HardwireConfig;

(* Network 27: LINMOT Code to use if using linear motor configuration Top folder *)
_e6(CLK := gIO.DOs.TopFolder);
_p7 := gFoldPushCtrlInterface.Status.LinMotConfig AND _e6.Q;
_p8 := _p7 AND gModeControlInterface.Commands.SetAutoMode;
_p9 := _p7 AND gModeControlInterface.Commands.SetJogMode;
IF _p8 OR _p9 THEN
    gFoldPushCtrlInterface.Parameters.LinMotTopFolder.Parameter.MpBasicParameters.Position := gFoldPushCtrlInterface.Parameters.LinMotTopFolder.Parameter.ExtendPos;
    gFoldPushCtrlInterface.Parameters.LinMotTopFolder.Command.MoveAbsoluteRequest := TRUE;
END_IF;

(* Network 28 *)
_p10 := gFoldPushCtrlInterface.Status.LinMotConfig AND gModeControlInterface.Commands.SetAutoMode;
_p11 := gFoldPushCtrlInterface.Status.LinMotConfig AND gModeControlInterface.Commands.SetJogMode;
_e12(CLK := gIO.DOs.TopFolder);
_e13(CLK := gRamCtrlInterface.Status.Running);
_p14 := (_p10 OR _p11) AND NOT gIO.DOs.TopFolder AND _e13.Q;
IF ((_p10 OR _p11) AND _e12.Q) OR _p14 THEN
    gFoldPushCtrlInterface.Parameters.LinMotTopFolder.Parameter.MpBasicParameters.Position := gFoldPushCtrlInterface.Parameters.LinMotTopFolder.Parameter.RetractPos;
    gFoldPushCtrlInterface.Parameters.LinMotTopFolder.Command.MoveAbsoluteRequest := TRUE;
END_IF;

(* Network 29: Bottom folder *)
_e15(CLK := gIO.DOs.BottomFolder);
_p16 := gFoldPushCtrlInterface.Status.LinMotConfig AND _e15.Q;
_p17 := _p16 AND gModeControlInterface.Commands.SetAutoMode;
_p18 := _p16 AND gModeControlInterface.Commands.SetJogMode;
IF _p17 OR _p18 THEN
    gFoldPushCtrlInterface.Parameters.LinMotBotFolder.Parameter.MpBasicParameters.Position := gFoldPushCtrlInterface.Parameters.LinMotBotFolder.Parameter.ExtendPos;
    gFoldPushCtrlInterface.Parameters.LinMotBotFolder.Command.MoveAbsoluteRequest := TRUE;
END_IF;

(* Network 30 *)
_p19 := gFoldPushCtrlInterface.Status.LinMotConfig AND gModeControlInterface.Commands.SetAutoMode;
_p20 := gFoldPushCtrlInterface.Status.LinMotConfig AND gModeControlInterface.Commands.SetJogMode;
_e21(CLK := gIO.DOs.BottomFolder);
_e22(CLK := gRamCtrlInterface.Status.Running);
_p23 := (_p19 OR _p20) AND NOT gIO.DOs.BottomFolder AND _e22.Q;
IF ((_p19 OR _p20) AND _e21.Q) OR _p23 THEN
    gFoldPushCtrlInterface.Parameters.LinMotBotFolder.Parameter.MpBasicParameters.Position := gFoldPushCtrlInterface.Parameters.LinMotBotFolder.Parameter.RetractPos;
    gFoldPushCtrlInterface.Parameters.LinMotBotFolder.Command.MoveAbsoluteRequest := TRUE;
END_IF;
END_PROGRAM
```

#### Variables.var - Local variables
```iecst
VAR
	Valve0OnBliss : BOOL;
	Valve2OnBliss : BOOL;
	Valve4OnBliss : BOOL;
	Valve6OnBliss : BOOL;
	Valve0OnNotBliss : BOOL;
	Valve2OnNotBliss : BOOL;
	Valve4OnNotBliss : BOOL;
	Valve6OnNotBliss : BOOL;
	DataSource : REAL;
END_VAR
```

### Program Logical/Actuators/VacuumControl (IEC)

#### Cyclic.ld - Cyclic code
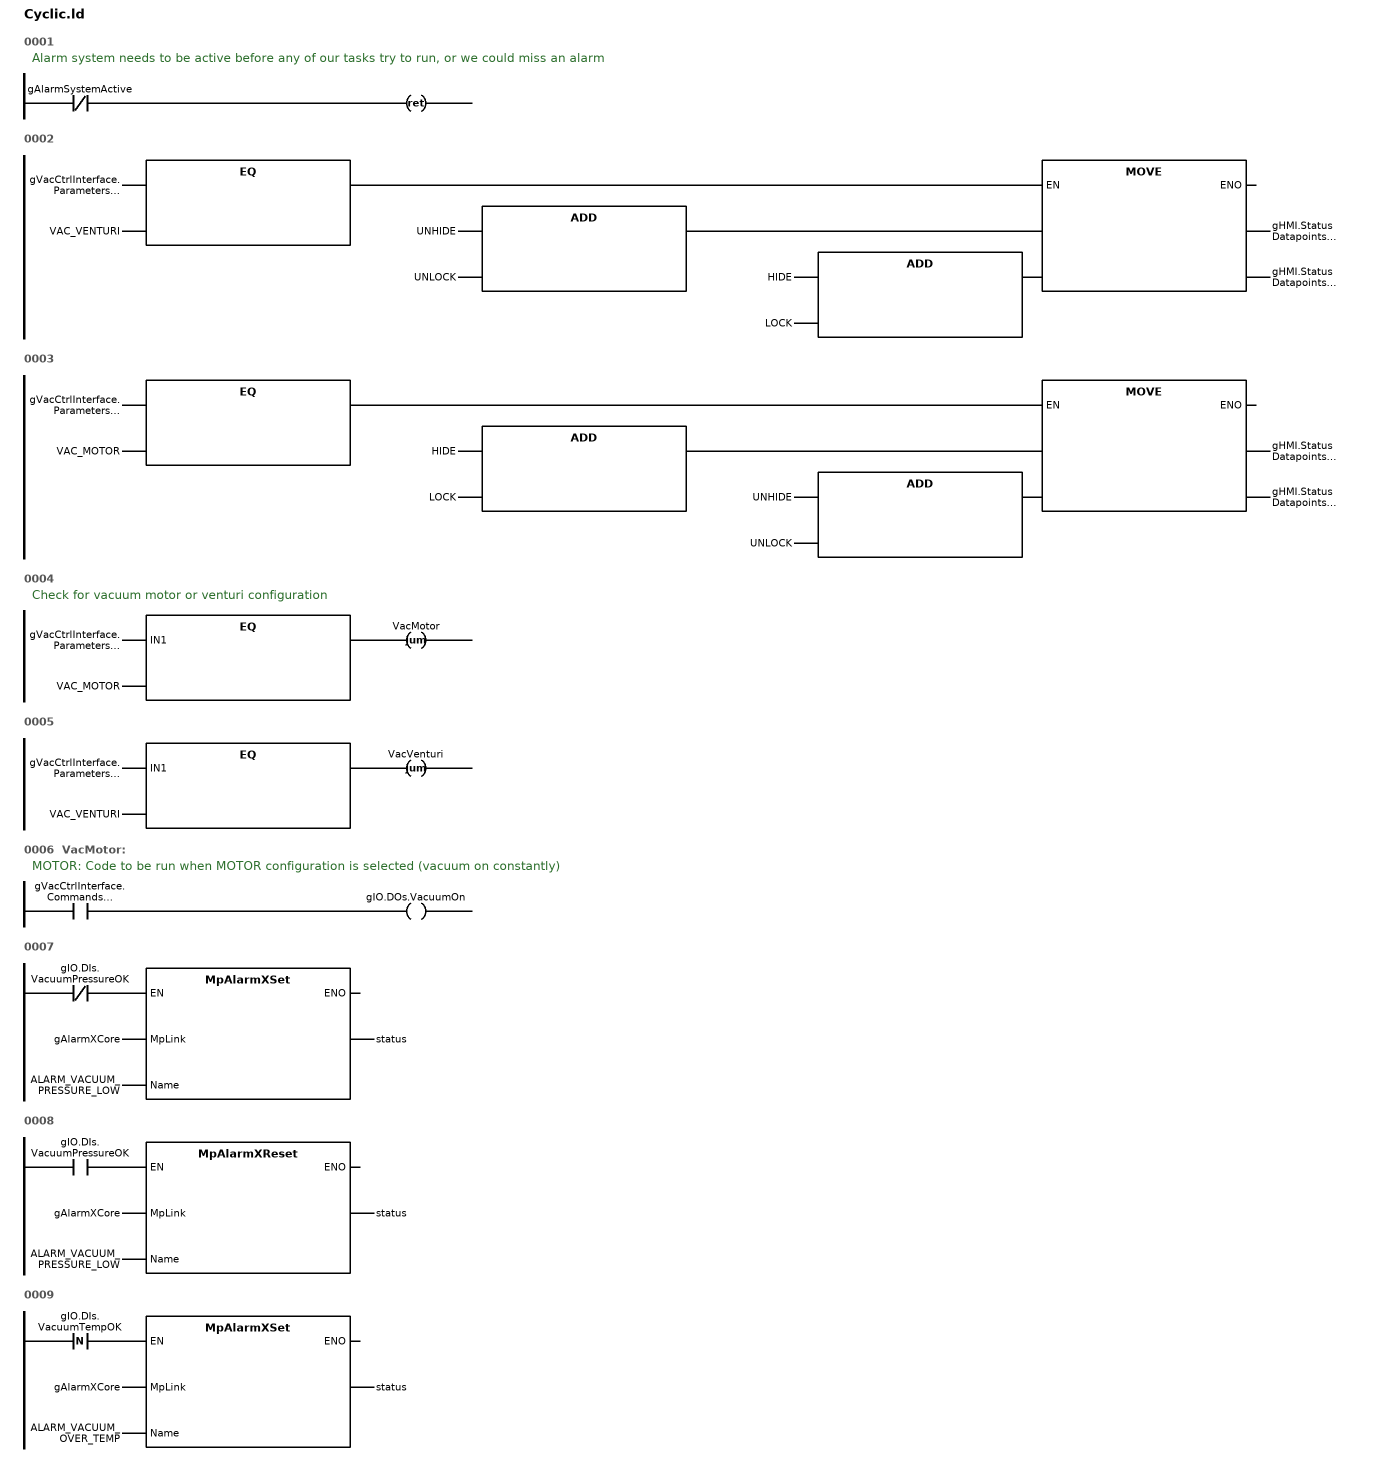
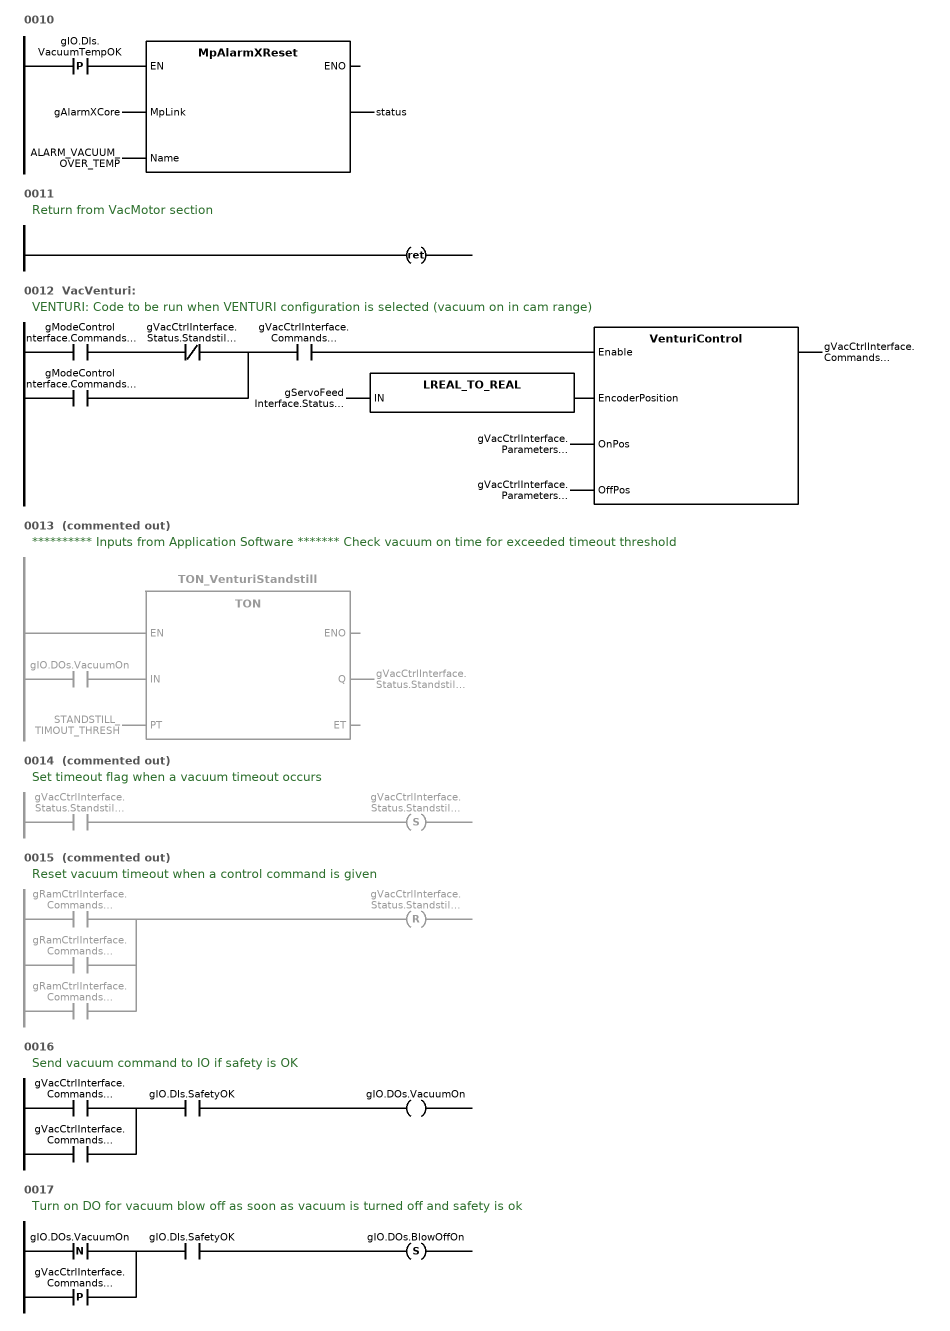
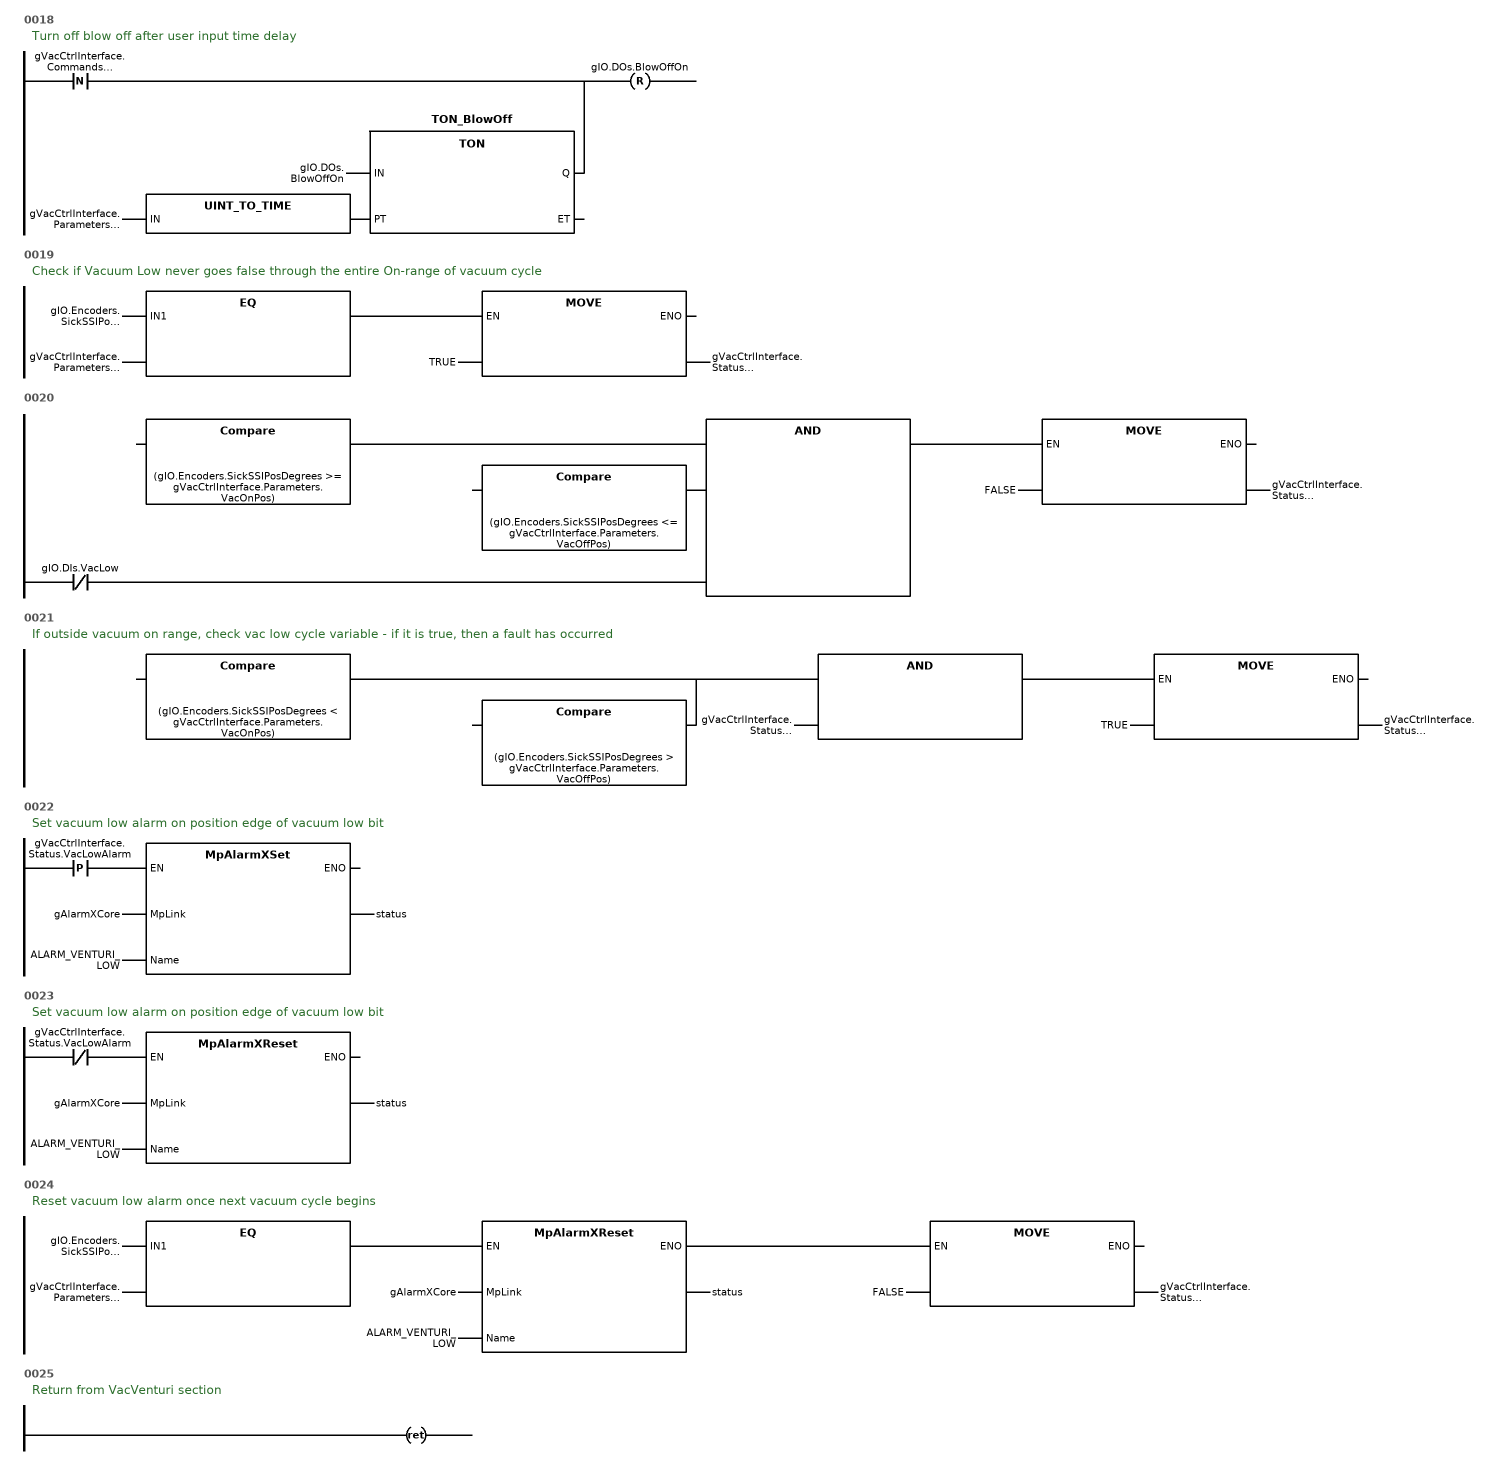
Ladder, written as Structured Text:
```iecst
PROGRAM _CYCLIC
VAR
    _t1 : BOOL;
    _t2 : BOOL;
    _e3 : F_TRIG;
    _e4 : R_TRIG;
    _e5 : F_TRIG;
    _e6 : R_TRIG;
    _e7 : F_TRIG;
    _p8 : BOOL;
    _p9 : BOOL;
    _p10 : BOOL;
    _e11 : R_TRIG;
    _p12 : BOOL;
    _p13 : BOOL;
END_VAR
(* Network 1: Alarm system needs to be active before any of our tasks try to run, or we could miss an alarm *)
IF NOT gAlarmSystemActive THEN RETURN; END_IF;

(* Network 2 *)
_t1 := gVacCtrlInterface.Parameters.VacConfig = VAC_VENTURI;
IF _t1 THEN
    gHMI.StatusDatapoints.VenturiVacuumSDP := UNHIDE + UNLOCK;
    gHMI.StatusDatapoints.MotorVacuumSDP := HIDE + LOCK;
END_IF;

(* Network 3 *)
_t2 := gVacCtrlInterface.Parameters.VacConfig = VAC_MOTOR;
IF _t2 THEN
    gHMI.StatusDatapoints.VenturiVacuumSDP := HIDE + LOCK;
    gHMI.StatusDatapoints.MotorVacuumSDP := UNHIDE + UNLOCK;
END_IF;

(* Network 4: Check for vacuum motor or venturi configuration *)
IF gVacCtrlInterface.Parameters.VacConfig = VAC_MOTOR THEN JMP VacMotor; END_IF;

(* Network 5 *)
IF gVacCtrlInterface.Parameters.VacConfig = VAC_VENTURI THEN JMP VacVenturi; END_IF;

(* Network 6: MOTOR: Code to be run when MOTOR configuration is selected (vacuum on constantly) *)
VacMotor:
gIO.DOs.VacuumOn := gVacCtrlInterface.Commands.VacuumOn;

(* Network 7 *)
IF NOT gIO.DIs.VacuumPressureOK THEN
    status := MpAlarmXSet(MpLink := gAlarmXCore, Name := ALARM_VACUUM_PRESSURE_LOW);
END_IF;

(* Network 8 *)
IF gIO.DIs.VacuumPressureOK THEN
    status := MpAlarmXReset(MpLink := gAlarmXCore, Name := ALARM_VACUUM_PRESSURE_LOW);
END_IF;

(* Network 9 *)
_e3(CLK := gIO.DIs.VacuumTempOK);
IF _e3.Q THEN status := MpAlarmXSet(MpLink := gAlarmXCore, Name := ALARM_VACUUM_OVER_TEMP); END_IF;

(* Network 10 *)
_e4(CLK := gIO.DIs.VacuumTempOK);
IF _e4.Q THEN status := MpAlarmXReset(MpLink := gAlarmXCore, Name := ALARM_VACUUM_OVER_TEMP); END_IF;

(* Network 11: Return from VacMotor section *)
RETURN;

(* Network 12: VENTURI: Code to be run when VENTURI configuration is selected (vacuum on in cam range) *)
VacVenturi:
gVacCtrlInterface.Commands.VenturiOn := VenturiControl(Enable := ((gModeControlInterface.Commands.SetAutoMode AND NOT gVacCtrlInterface.Status.StandstillTimoutSet) OR gModeControlInterface.Commands.SetJogMode) AND gVacCtrlInterface.Commands.VacuumOn, EncoderPosition := LREAL_TO_REAL(gServoFeedInterface.Status.ActualPosition), OnPos := gVacCtrlInterface.Parameters.VacOnPos, OffPos := gVacCtrlInterface.Parameters.VacOffPos);

(* Network 13:  ********** Inputs from Application Software ******* Check vacuum on time for exceeded timeout threshold *) (* commented out *)
// TON_VenturiStandstill(IN := gIO.DOs.VacuumOn, PT := STANDSTILL_TIMOUT_THRESH);
// gVacCtrlInterface.Status.StandstillTimout := TON_VenturiStandstill.Q;

(* Network 14: Set timeout flag when a vacuum timeout occurs *) (* commented out *)
// IF gVacCtrlInterface.Status.StandstillTimout THEN
//     gVacCtrlInterface.Status.StandstillTimoutSet := TRUE;
// END_IF;

(* Network 15: Reset vacuum timeout when a control command is given *) (* commented out *)
// IF gRamCtrlInterface.Commands.JogPositive OR gRamCtrlInterface.Commands.JogNegative OR gRamCtrlInterface.Commands.MoveVelocity THEN
//     gVacCtrlInterface.Status.StandstillTimoutSet := FALSE;
// END_IF;

(* Network 16: Send vacuum command to IO if safety is OK *)
gIO.DOs.VacuumOn := (gVacCtrlInterface.Commands.VenturiOn OR gVacCtrlInterface.Commands.VenturiOnManual) AND gIO.DIs.SafetyOK;

(* Network 17: Turn on DO for vacuum blow off as soon as vacuum is turned off and safety is ok *)
_e5(CLK := gIO.DOs.VacuumOn);
_e6(CLK := gVacCtrlInterface.Commands.BlowOffOnManual);
IF (_e5.Q OR _e6.Q) AND gIO.DIs.SafetyOK THEN gIO.DOs.BlowOffOn := TRUE; END_IF;

(* Network 18: Turn off blow off after user input time delay *)
_e7(CLK := gVacCtrlInterface.Commands.BlowOffOnManual);
IF _e7.Q OR TON_BlowOff.Q THEN gIO.DOs.BlowOffOn := FALSE; END_IF;
TON_BlowOff(IN := gIO.DOs.BlowOffOn, PT := UINT_TO_TIME(gVacCtrlInterface.Parameters.BlowOffTime));

(* Network 19: Check if Vacuum Low never goes false through the entire On-range of vacuum cycle *)
_p8 := gIO.Encoders.SickSSIPosDegrees = gVacCtrlInterface.Parameters.VacOnPos;
IF _p8 THEN gVacCtrlInterface.Status.VacLowCycle := TRUE; END_IF;

(* Network 20 *)
_p9 := ((gIO.Encoders.SickSSIPosDegrees >= gVacCtrlInterface.Parameters.VacOnPos)) AND ((gIO.Encoders.SickSSIPosDegrees <= gVacCtrlInterface.Parameters.VacOffPos)) AND NOT gIO.DIs.VacLow;
IF _p9 THEN gVacCtrlInterface.Status.VacLowCycle := FALSE; END_IF;

(* Network 21: If outside vacuum on range, check vac low cycle variable - if it is true, then a fault has occurred *)
_p10 := (((gIO.Encoders.SickSSIPosDegrees < gVacCtrlInterface.Parameters.VacOnPos)) OR ((gIO.Encoders.SickSSIPosDegrees > gVacCtrlInterface.Parameters.VacOffPos))) AND gVacCtrlInterface.Status.VacLowCycle;
IF _p10 THEN gVacCtrlInterface.Status.VacLowAlarm := TRUE; END_IF;

(* Network 22: Set vacuum low alarm on position edge of vacuum low bit *)
_e11(CLK := gVacCtrlInterface.Status.VacLowAlarm);
IF _e11.Q THEN status := MpAlarmXSet(MpLink := gAlarmXCore, Name := ALARM_VENTURI_LOW); END_IF;

(* Network 23: Set vacuum low alarm on position edge of vacuum low bit *)
_p12 := NOT gVacCtrlInterface.Status.VacLowAlarm;
IF _p12 THEN status := MpAlarmXReset(MpLink := gAlarmXCore, Name := ALARM_VENTURI_LOW); END_IF;

(* Network 24: Reset vacuum low alarm once next vacuum cycle begins *)
IF gIO.Encoders.SickSSIPosDegrees = gVacCtrlInterface.Parameters.VacOnPos THEN
    status := MpAlarmXReset(MpLink := gAlarmXCore, Name := ALARM_VENTURI_LOW);
END_IF;
_p13 := gIO.Encoders.SickSSIPosDegrees = gVacCtrlInterface.Parameters.VacOnPos;
IF _p13 THEN gVacCtrlInterface.Status.VacLowAlarm := FALSE; END_IF;

(* Network 25: Return from VacVenturi section *)
RETURN;
END_PROGRAM
```

#### Init.st
```iecst
PROGRAM _INIT

	IF(gVacCtrlInterface.Parameters.BlowOffTime < 100) THEN
		gVacCtrlInterface.Parameters.BlowOffTime := 100;
	END_IF

END_PROGRAM
```

#### Variables.var - Local variables
```iecst
VAR
	status : UDINT;
	TON_BlowOff : TON; (*Timer for blow off after vacuum is shut off (user defined time)*)
END_VAR
VAR CONSTANT
	STANDSTILL_TIMOUT_THRESH : TIME := T#15s;
END_VAR
VAR
	TON_VenturiStandstill : TON;
END_VAR
```

### Program Logical/Actuators/NordsonComm/NordsonMBComm (IEC)
